LIN {X 0,Y 488.421,Z 680.985,A -85,B 0,C 180,E1 -6398.273,E2 -6398.273} C_VEL
LIN {X 0,Y 488.699,Z 673.076,A -85,B 0,C 180,E1 -6399.52,E2 -6399.52} C_VEL
LIN {X 0,Y 489.009,Z 665.001,A -85,B 0,C 180,E1 -6400.559,E2 -6400.559} C_VEL
LIN {X 0,Y 489.51,Z 655.097,A -85,B 0,C 180,E1 -6401.596,E2 -6401.596} C_VEL
LIN {X 0,Y 489.842,Z 643.67,A -85,B 0,C 180,E1 -6402.557,E2 -6402.557} C_VEL
LIN {X 0,Y 490.248,Z 633.111,A -85,B 0,C 180,E1 -6403.26,E2 -6403.26} C_VEL
LIN {X 0,Y 490.638,Z 620.98,A -85,B 0,C 180,E1 -6403.883,E2 -6403.883} C_VEL
LIN {X 0,Y 490.956,Z 608.45,A -85,B 0,C 180,E1 -6404.349,E2 -6404.349} C_VEL
LIN {X 0,Y 491.208,Z 595.654,A -85,B 0,C 180,E1 -6404.659,E2 -6404.659} C_VEL
LIN {X 0,Y 491.628,Z 499.894,A -85,B 0,C 180,E1 -6406.077,E2 -6406.077} C_VEL
LIN {X 0,Y 489.945,Z 488.116,A -85,B 0,C 180,E1 -6406.322,E2 -6406.322} C_VEL
LIN {X 0,Y 490.166,Z 476.152,A -85,B 0,C 180,E1 -6407.739,E2 -6407.739} C_VEL
LIN {X 0,Y 490.799,Z 452.084,A -85,B 0,C 180,E1 -6410.757,E2 -6410.757} C_VEL
LIN {X 0,Y 491.628,Z 428.446,A -85,B 0,C 180,E1 -6413.807,E2 -6413.807} C_VEL
LIN {X 0,Y 492.314,Z 404.124,A -85,B 0,C 180,E1 -6416.952,E2 -6416.952} C_VEL
LIN {X 0,Y 490.804,Z 396.546,A -85,B 0,C 180,E1 -6418.011,E2 -6418.011} C_VEL
LIN {X 0,Y 488.774,Z 387.78,A -85,B 0,C 180,E1 -6419.267,E2 -6419.267} C_VEL
LIN {X 0,Y 488.706,Z 387.61,A -85,B 0,C 180,E1 -6422.147,E2 -6422.147} C_VEL
LIN {X 0,Y 488.713,Z 387.61,A -85,B 0,C 180,E1 -6425.116,E2 -6425.116} C_VEL
LIN {X 0,Y 488.66,Z 387.615,A -85,B 0,C 180,E1 -6428.202,E2 -6428.202} C_VEL
LIN {X 0,Y 488.696,Z 387.602,A -85,B 0,C 180,E1 -6430.341,E2 -6430.341} C_VEL
LIN {X 0,Y 488.676,Z 387.609,A -85,B 0,C 180,E1 -6433.656,E2 -6433.656} C_VEL
LIN {X 0,Y 488.678,Z 387.61,A -85,B 0,C 180,E1 -6436.344,E2 -6436.344} C_VEL
LIN {X 0,Y 488.707,Z 387.611,A -85,B 0,C 180,E1 -6439.674,E2 -6439.674} C_VEL
LIN {X 0,Y 488.662,Z 387.607,A -85,B 0,C 180,E1 -6442.839,E2 -6442.839} C_VEL
LIN {X 0,Y 488.721,Z 387.604,A -85,B 0,C 180,E1 -6445.886,E2 -6445.886} C_VEL
LIN {X 0,Y 488.693,Z 387.608,A -85,B 0,C 180,E1 -6448.82,E2 -6448.82} C_VEL
LIN {X 0,Y 488.695,Z 387.608,A -85,B 0,C 180,E1 -6451.668,E2 -6451.668} C_VEL
LIN {X 0,Y 488.702,Z 387.606,A -85,B 0,C 180,E1 -6454.959,E2 -6454.959} C_VEL
LIN {X 0,Y 488.7,Z 387.61,A -85,B 0,C 180,E1 -6458.043,E2 -6458.043} C_VEL
LIN {X 0,Y 488.734,Z 387.6,A -85,B 0,C 180,E1 -6460.686,E2 -6460.686} C_VEL
LIN {X 0,Y 488.714,Z 387.607,A -85,B 0,C 180,E1 -6464.143,E2 -6464.143} C_VEL
LIN {X 0,Y 488.725,Z 387.601,A -85,B 0,C 180,E1 -6466.698,E2 -6466.698} C_VEL
LIN {X 0,Y 488.704,Z 387.598,A -85,B 0,C 180,E1 -6469.225,E2 -6469.225} C_VEL
LIN {X 0,Y 488.763,Z 387.606,A -85,B 0,C 180,E1 -6471.733,E2 -6471.733} C_VEL
LIN {X 0,Y 488.816,Z 387.587,A -85,B 0,C 180,E1 -6474.224,E2 -6474.224} C_VEL
LIN {X 0,Y 488.944,Z 387.576,A -85,B 0,C 180,E1 -6477.529,E2 -6477.529} C_VEL
LIN {X 0,Y 488.945,Z 387.578,A -85,B 0,C 180,E1 -6480,E2 -6480} C_VEL
LIN {X 0,Y 488.945,Z 387.566,A -85,B 0,C 180,E1 -6482.471,E2 -6482.471} C_VEL
LIN {X 0,Y 488.814,Z 387.599,A -85,B 0,C 180,E1 -6485.776,E2 -6485.776} C_VEL
LIN {X 0,Y 488.76,Z 387.595,A -85,B 0,C 180,E1 -6488.267,E2 -6488.267} C_VEL
LIN {X 0,Y 488.788,Z 387.596,A -85,B 0,C 180,E1 -6491.613,E2 -6491.613} C_VEL
LIN {X 0,Y 488.723,Z 387.601,A -85,B 0,C 180,E1 -6495.002,E2 -6495.002} C_VEL
LIN {X 0,Y 488.705,Z 387.606,A -85,B 0,C 180,E1 -6498.444,E2 -6498.444} C_VEL
LIN {X 0,Y 488.682,Z 387.608,A -85,B 0,C 180,E1 -6501.072,E2 -6501.072} C_VEL
LIN {X 0,Y 488.667,Z 387.608,A -85,B 0,C 180,E1 -6503.747,E2 -6503.747} C_VEL
LIN {X 0,Y 488.671,Z 387.611,A -85,B 0,C 180,E1 -6506.477,E2 -6506.477} C_VEL
LIN {X 0,Y 488.702,Z 387.6,A -85,B 0,C 180,E1 -6509.272,E2 -6509.272} C_VEL
LIN {X 0,Y 488.692,Z 387.611,A -85,B 0,C 180,E1 -6512.148,E2 -6512.148} C_VEL
LIN {X 0,Y 488.708,Z 387.601,A -85,B 0,C 180,E1 -6515.116,E2 -6515.116} C_VEL
LIN {X 0,Y 488.651,Z 387.612,A -85,B 0,C 180,E1 -6518.203,E2 -6518.203} C_VEL
LIN {X 0,Y 488.644,Z 387.595,A -85,B 0,C 180,E1 -6521.422,E2 -6521.422} C_VEL
LIN {X 0,Y 488.698,Z 387.607,A -85,B 0,C 180,E1 -6524.803,E2 -6524.803} C_VEL
LIN {X 0,Y 488.65,Z 387.613,A -85,B 0,C 180,E1 -6527.469,E2 -6527.469} C_VEL
LIN {X 0,Y 488.671,Z 387.608,A -85,B 0,C 180,E1 -6530.742,E2 -6530.742} C_VEL
LIN {X 0,Y 488.642,Z 387.622,A -85,B 0,C 180,E1 -6533.864,E2 -6533.864} C_VEL
LIN {X 0,Y 488.694,Z 387.611,A -85,B 0,C 180,E1 -6536.523,E2 -6536.523} C_VEL
LIN {X 0,Y 488.666,Z 387.618,A -85,B 0,C 180,E1 -6539.776,E2 -6539.776} C_VEL
LIN {X 0,Y 488.734,Z 387.967,A -85,B 0,C 180,E1 -6540.138,E2 -6540.138} C_VEL
LIN {X 0,Y 492.353,Z 403.874,A -85,B 0,C 180,E1 -6542.467,E2 -6542.467} C_VEL
LIN {X 0,Y 491.871,Z 419.05,A -85,B 0,C 180,E1 -6544.452,E2 -6544.452} C_VEL
LIN {X 0,Y 490.95,Z 442.63,A -85,B 0,C 180,E1 -6547.485,E2 -6547.485} C_VEL
LIN {X 0,Y 490.174,Z 466.628,A -85,B 0,C 180,E1 -6550.527,E2 -6550.527} C_VEL
LIN {X 0,Y 489.479,Z 492.055,A -85,B 0,C 180,E1 -6553.698,E2 -6553.698} C_VEL
LIN {X 0,Y 491.532,Z 510.881,A -85,B 0,C 180,E1 -6554.093,E2 -6554.093} C_VEL
LIN {X 0,Y 490.766,Z 603.473,A -85,B 0,C 180,E1 -6555.566,E2 -6555.566} C_VEL
LIN {X 0,Y 490.386,Z 620.377,A -85,B 0,C 180,E1 -6556.031,E2 -6556.031} C_VEL
LIN {X 0,Y 490.093,Z 633.651,A -85,B 0,C 180,E1 -6556.577,E2 -6556.577} C_VEL
LIN {X 0,Y 489.785,Z 644.595,A -85,B 0,C 180,E1 -6557.191,E2 -6557.191} C_VEL
LIN {X 0,Y 489.453,Z 655.726,A -85,B 0,C 180,E1 -6557.992,E2 -6557.992} C_VEL
LIN {X 0,Y 489.043,Z 666.053,A -85,B 0,C 180,E1 -6558.918,E2 -6558.918} C_VEL
LIN {X 0,Y 488.789,Z 674.567,A -85,B 0,C 180,E1 -6559.855,E2 -6559.855} C_VEL
LIN {X 0,Y 488.508,Z 682.384,A -85,B 0,C 180,E1 -6560.894,E2 -6560.894} C_VEL
LIN {X 0,Y 488.295,Z 689.986,A -85,B 0,C 180,E1 -6562.141,E2 -6562.141} C_VEL
LIN {X 0,Y 488.105,Z 696.43,A -85,B 0,C 180,E1 -6563.465,E2 -6563.465} C_VEL
LIN {X 0,Y 488.086,Z 700.893,A -85,B 0,C 180,E1 -6564.629,E2 -6564.629} C_VEL
LIN {X 0,Y 488.026,Z 704.563,A -85,B 0,C 180,E1 -6565.871,E2 -6565.871} C_VEL
LIN {X 0,Y 488.028,Z 706.453,A -85,B 0,C 180,E1 -6566.698,E2 -6566.698} C_VEL
LIN {X 0,Y 487.974,Z 707.88,A -85,B 0,C 180,E1 -6567.524,E2 -6567.524} C_VEL
LIN {X 0,Y 487.953,Z 708.886,A -85,B 0,C 180,E1 -6568.349,E2 -6568.349} C_VEL
LIN {X 0,Y 487.921,Z 709.721,A -85,B 0,C 180,E1 -6570,E2 -6570} C_VEL
LIN {X 0,Y 487.933,Z 709.501,A -85,B 0,C 180,E1 -6570.825,E2 -6570.825} C_VEL
LIN {X 0,Y 487.958,Z 708.887,A -85,B 0,C 180,E1 -6571.651,E2 -6571.651} C_VEL
LIN {X 0,Y 487.983,Z 707.882,A -85,B 0,C 180,E1 -6572.476,E2 -6572.476} C_VEL
LIN {X 0,Y 488.037,Z 706.455,A -85,B 0,C 180,E1 -6573.302,E2 -6573.302} C_VEL
LIN {X 0,Y 488.016,Z 703.483,A -85,B 0,C 180,E1 -6574.543,E2 -6574.543} C_VEL
LIN {X 0,Y 488.108,Z 699.445,A -85,B 0,C 180,E1 -6575.785,E2 -6575.785} C_VEL
LIN {X 0,Y 488.184,Z 693.211,A -85,B 0,C 180,E1 -6577.237,E2 -6577.237} C_VEL
LIN {X 0,Y 488.42,Z 686.403,A -85,B 0,C 180,E1 -6578.481,E2 -6578.481} C_VEL
LIN {X 0,Y 488.571,Z 679.428,A -85,B 0,C 180,E1 -6579.522,E2 -6579.522} C_VEL
LIN {X 0,Y 488.879,Z 670.989,A -85,B 0,C 180,E1 -6580.561,E2 -6580.561} C_VEL
LIN {X 0,Y 489.254,Z 660.526,A -85,B 0,C 180,E1 -6581.602,E2 -6581.602} C_VEL
LIN {X 0,Y 489.587,Z 650.136,A -85,B 0,C 180,E1 -6582.435,E2 -6582.435} C_VEL
LIN {X 0,Y 489.928,Z 638.639,A -85,B 0,C 180,E1 -6583.163,E2 -6583.163} C_VEL
LIN {X 0,Y 490.285,Z 626.638,A -85,B 0,C 180,E1 -6583.734,E2 -6583.734} C_VEL
LIN {X 0,Y 490.503,Z 614.471,A -85,B 0,C 180,E1 -6584.151,E2 -6584.151} C_VEL
LIN {X 0,Y 490.732,Z 602.483,A -85,B 0,C 180,E1 -6584.409,E2 -6584.409} C_VEL
LIN {X 0,Y 491.382,Z 509.881,A -85,B 0,C 180,E1 -6585.871,E2 -6585.871} C_VEL
LIN {X 0,Y 489.25,Z 488.746,A -85,B 0,C 180,E1 -6586.327,E2 -6586.327} C_VEL
LIN {X 0,Y 489.772,Z 466.119,A -85,B 0,C 180,E1 -6589.098,E2 -6589.098} C_VEL
LIN {X 0,Y 490.419,Z 442.199,A -85,B 0,C 180,E1 -6592.097,E2 -6592.097} C_VEL
LIN {X 0,Y 491.22,Z 418.158,A -85,B 0,C 180,E1 -6595.191,E2 -6595.191} C_VEL
LIN {X 0,Y 491.802,Z 402.9,A -85,B 0,C 180,E1 -6597.212,E2 -6597.212} C_VEL
LIN {X 0,Y 489.495,Z 391.112,A -85,B 0,C 180,E1 -6598.972,E2 -6598.972} C_VEL
LIN {X 0,Y 488.701,Z 387.728,A -85,B 0,C 180,E1 -6599.538,E2 -6599.538} C_VEL
LIN {X 0,Y 488.679,Z 387.616,A -85,B 0,C 180,E1 -6602.149,E2 -6602.149} C_VEL
LIN {X 0,Y 488.696,Z 387.611,A -85,B 0,C 180,E1 -6605.117,E2 -6605.117} C_VEL
LIN {X 0,Y 488.65,Z 387.619,A -85,B 0,C 180,E1 -6608.203,E2 -6608.203} C_VEL
LIN {X 0,Y 488.644,Z 387.618,A -85,B 0,C 180,E1 -6611.422,E2 -6611.422} C_VEL
LIN {X 0,Y 488.702,Z 387.608,A -85,B 0,C 180,E1 -6614.803,E2 -6614.803} C_VEL
LIN {X 0,Y 488.651,Z 387.617,A -85,B 0,C 180,E1 -6617.47,E2 -6617.47} C_VEL
LIN {X 0,Y 488.705,Z 387.612,A -85,B 0,C 180,E1 -6619.674,E2 -6619.674} C_VEL
LIN {X 0,Y 488.662,Z 387.613,A -85,B 0,C 180,E1 -6622.839,E2 -6622.839} C_VEL
LIN {X 0,Y 488.725,Z 387.609,A -85,B 0,C 180,E1 -6625.887,E2 -6625.887} C_VEL
LIN {X 0,Y 488.694,Z 387.61,A -85,B 0,C 180,E1 -6628.82,E2 -6628.82} C_VEL
LIN {X 0,Y 488.714,Z 387.612,A -85,B 0,C 180,E1 -6631.669,E2 -6631.669} C_VEL
LIN {X 0,Y 488.707,Z 387.606,A -85,B 0,C 180,E1 -6634.442,E2 -6634.442} C_VEL
LIN {X 0,Y 488.724,Z 387.61,A -85,B 0,C 180,E1 -6637.153,E2 -6637.153} C_VEL
LIN {X 0,Y 488.728,Z 387.609,A -85,B 0,C 180,E1 -6639.811,E2 -6639.811} C_VEL
LIN {X 0,Y 488.718,Z 387.61,A -85,B 0,C 180,E1 -6642.423,E2 -6642.423} C_VEL
LIN {X 0,Y 488.774,Z 387.749,A -85,B 0,C 180,E1 -6644.092,E2 -6644.092} C_VEL
LIN {X 0,Y 488.957,Z 388.568,A -85,B 0,C 180,E1 -6644.226,E2 -6644.226} C_VEL
LIN {X 0,Y 491.703,Z 396.705,A -85,B 0,C 180,E1 -6644.497,E2 -6644.497} C_VEL
LIN {X 0,Y 491.048,Z 471.478,A -85,B 0,C 180,E1 -6645.76,E2 -6645.76} C_VEL
LIN {X 0,Y 490.918,Z 485.433,A -85,B 0,C 180,E1 -6646.178,E2 -6646.178} C_VEL
LIN {X 0,Y 490.785,Z 498.232,A -85,B 0,C 180,E1 -6646.755,E2 -6646.755} C_VEL
LIN {X 0,Y 490.578,Z 510.162,A -85,B 0,C 180,E1 -6647.475,E2 -6647.475} C_VEL
LIN {X 0,Y 490.245,Z 521.111,A -85,B 0,C 180,E1 -6648.317,E2 -6648.317} C_VEL
LIN {X 0,Y 489.959,Z 530.794,A -85,B 0,C 180,E1 -6649.253,E2 -6649.253} C_VEL
LIN {X 0,Y 489.7,Z 539.557,A -85,B 0,C 180,E1 -6650.292,E2 -6650.292} C_VEL
LIN {X 0,Y 489.412,Z 546.759,A -85,B 0,C 180,E1 -6651.328,E2 -6651.328} C_VEL
LIN {X 0,Y 489.082,Z 553.808,A -85,B 0,C 180,E1 -6652.569,E2 -6652.569} C_VEL
LIN {X 0,Y 488.992,Z 559.358,A -85,B 0,C 180,E1 -6653.812,E2 -6653.812} C_VEL
LIN {X 0,Y 488.733,Z 563.713,A -85,B 0,C 180,E1 -6655.05,E2 -6655.05} C_VEL
LIN {X 0,Y 488.65,Z 565.979,A -85,B 0,C 180,E1 -6655.876,E2 -6655.876} C_VEL
LIN {X 0,Y 488.703,Z 567.797,A -85,B 0,C 180,E1 -6656.702,E2 -6656.702} C_VEL
LIN {X 0,Y 488.561,Z 569.208,A -85,B 0,C 180,E1 -6657.527,E2 -6657.527} C_VEL
LIN {X 0,Y 488.58,Z 570.15,A -85,B 0,C 180,E1 -6658.351,E2 -6658.351} C_VEL
LIN {X 0,Y 488.487,Z 570.885,A -85,B 0,C 180,E1 -6660,E2 -6660} C_VEL
LIN {X 0,Y 488.504,Z 570.624,A -85,B 0,C 180,E1 -6660.824,E2 -6660.824} C_VEL
LIN {X 0,Y 488.438,Z 569.968,A -85,B 0,C 180,E1 -6661.649,E2 -6661.649} C_VEL
LIN {X 0,Y 488.535,Z 568.897,A -85,B 0,C 180,E1 -6662.474,E2 -6662.474} C_VEL
LIN {X 0,Y 488.495,Z 567.446,A -85,B 0,C 180,E1 -6663.299,E2 -6663.299} C_VEL
LIN {X 0,Y 488.648,Z 564.404,A -85,B 0,C 180,E1 -6664.537,E2 -6664.537} C_VEL
LIN {X 0,Y 488.745,Z 560.322,A -85,B 0,C 180,E1 -6665.777,E2 -6665.777} C_VEL
LIN {X 0,Y 488.981,Z 554.834,A -85,B 0,C 180,E1 -6667.061,E2 -6667.061} C_VEL
LIN {X 0,Y 489.212,Z 547.178,A -85,B 0,C 180,E1 -6668.468,E2 -6668.468} C_VEL
LIN {X 0,Y 489.485,Z 540.175,A -85,B 0,C 180,E1 -6669.504,E2 -6669.504} C_VEL
LIN {X 0,Y 489.681,Z 531.737,A -85,B 0,C 180,E1 -6670.544,E2 -6670.544} C_VEL
LIN {X 0,Y 489.989,Z 521.287,A -85,B 0,C 180,E1 -6671.584,E2 -6671.584} C_VEL
LIN {X 0,Y 490.392,Z 509.565,A -85,B 0,C 180,E1 -6672.512,E2 -6672.512} C_VEL
LIN {X 0,Y 490.542,Z 497.636,A -85,B 0,C 180,E1 -6673.252,E2 -6673.252} C_VEL
LIN {X 0,Y 490.776,Z 485.334,A -85,B 0,C 180,E1 -6673.826,E2 -6673.826} C_VEL
LIN {X 0,Y 490.962,Z 472.814,A -85,B 0,C 180,E1 -6674.243,E2 -6674.243} C_VEL
LIN {X 0,Y 491.012,Z 458.482,A -85,B 0,C 180,E1 -6674.533,E2 -6674.533} C_VEL
LIN {X 0,Y 491.417,Z 395.815,A -85,B 0,C 180,E1 -6675.535,E2 -6675.535} C_VEL
LIN {X 0,Y 488.913,Z 388.41,A -85,B 0,C 180,E1 -6675.764,E2 -6675.764} C_VEL
LIN {X 0,Y 488.774,Z 387.692,A -85,B 0,C 180,E1 -6675.908,E2 -6675.908} C_VEL
LIN {X 0,Y 488.745,Z 387.605,A -85,B 0,C 180,E1 -6679.313,E2 -6679.313} C_VEL
LIN {X 0,Y 488.701,Z 387.608,A -85,B 0,C 180,E1 -6681.957,E2 -6681.957} C_VEL
LIN {X 0,Y 488.734,Z 387.607,A -85,B 0,C 180,E1 -6685.049,E2 -6685.049} C_VEL
LIN {X 0,Y 488.709,Z 387.603,A -85,B 0,C 180,E1 -6687.399,E2 -6687.399} C_VEL
LIN {X 0,Y 488.712,Z 387.605,A -85,B 0,C 180,E1 -6690.363,E2 -6690.363} C_VEL
LIN {X 0,Y 488.732,Z 387.597,A -85,B 0,C 180,E1 -6693.483,E2 -6693.483} C_VEL
LIN {X 0,Y 488.683,Z 387.612,A -85,B 0,C 180,E1 -6696.354,E2 -6696.354} C_VEL
LIN {X 0,Y 488.703,Z 387.608,A -85,B 0,C 180,E1 -6699.254,E2 -6699.254} C_VEL
LIN {X 0,Y 488.69,Z 387.61,A -85,B 0,C 180,E1 -6702.526,E2 -6702.526} C_VEL
LIN {X 0,Y 488.703,Z 387.606,A -85,B 0,C 180,E1 -6705.197,E2 -6705.197} C_VEL
LIN {X 0,Y 488.697,Z 387.612,A -85,B 0,C 180,E1 -6708.583,E2 -6708.583} C_VEL
LIN {X 0,Y 488.703,Z 387.6,A -85,B 0,C 180,E1 -6710.948,E2 -6710.948} C_VEL
LIN {X 0,Y 488.666,Z 387.613,A -85,B 0,C 180,E1 -6713.462,E2 -6713.462} C_VEL
LIN {X 0,Y 488.026,Z 387.695,A -85,B 0,C 180,E1 -6714.15,E2 -6714.15} C_VEL
LIN {X 0,Y 485.191,Z 388.045,A -85,B 0,C 180,E1 -6715.267,E2 -6715.267} C_VEL
LIN {X 0,Y 482.782,Z 388.347,A -85,B 0,C 180,E1 -6716.167,E2 -6716.167} C_VEL
LIN {X 0,Y 481.751,Z 388.474,A -85,B 0,C 180,E1 -6716.863,E2 -6716.863} C_VEL
LIN {X 0,Y 481.67,Z 388.481,A -85,B 0,C 180,E1 -6717.098,E2 -6717.098} C_VEL
LIN {X 0,Y 481.734,Z 388.669,A -85,B 0,C 180,E1 -6720.575,E2 -6720.575} C_VEL
LIN {X 0,Y 485.358,Z 404.631,A -85,B 0,C 180,E1 -6722.863,E2 -6722.863} C_VEL
LIN {X 0,Y 485.19,Z 415.109,A -85,B 0,C 180,E1 -6724.243,E2 -6724.243} C_VEL
LIN {X 0,Y 484.486,Z 435.748,A -85,B 0,C 180,E1 -6726.942,E2 -6726.942} C_VEL
LIN {X 0,Y 483.714,Z 457.932,A -85,B 0,C 180,E1 -6729.814,E2 -6729.814} C_VEL
LIN {X 0,Y 483.09,Z 482.393,A -85,B 0,C 180,E1 -6732.867,E2 -6732.867} C_VEL
LIN {X 0,Y 482.979,Z 488.109,A -85,B 0,C 180,E1 -6733.531,E2 -6733.531} C_VEL
LIN {X 0,Y 484.947,Z 502.633,A -85,B 0,C 180,E1 -6733.829,E2 -6733.829} C_VEL
LIN {X 0,Y 484.243,Z 598.949,A -85,B 0,C 180,E1 -6735.287,E2 -6735.287} C_VEL
LIN {X 0,Y 483.985,Z 612.191,A -85,B 0,C 180,E1 -6735.655,E2 -6735.655} C_VEL
LIN {X 0,Y 483.6,Z 624.672,A -85,B 0,C 180,E1 -6736.18,E2 -6736.18} C_VEL
LIN {X 0,Y 483.21,Z 636.877,A -85,B 0,C 180,E1 -6736.873,E2 -6736.873} C_VEL
LIN {X 0,Y 482.826,Z 648.198,A -85,B 0,C 180,E1 -6737.709,E2 -6737.709} C_VEL
LIN {X 0,Y 482.267,Z 659.494,A -85,B 0,C 180,E1 -6738.76,E2 -6738.76} C_VEL
LIN {X 0,Y 481.957,Z 667.756,A -85,B 0,C 180,E1 -6739.71,E2 -6739.71} C_VEL
LIN {X 0,Y 481.604,Z 675.394,A -85,B 0,C 180,E1 -6740.763,E2 -6740.763} C_VEL
LIN {X 0,Y 481.31,Z 682.842,A -85,B 0,C 180,E1 -6742.026,E2 -6742.026} C_VEL
LIN {X 0,Y 481.117,Z 689.192,A -85,B 0,C 180,E1 -6743.377,E2 -6743.377} C_VEL
LIN {X 0,Y 481.009,Z 693.557,A -85,B 0,C 180,E1 -6744.55,E2 -6744.55} C_VEL
LIN {X 0,Y 480.88,Z 697.183,A -85,B 0,C 180,E1 -6745.81,E2 -6745.81} C_VEL
LIN {X 0,Y 480.899,Z 699.049,A -85,B 0,C 180,E1 -6746.649,E2 -6746.649} C_VEL
LIN {X 0,Y 480.824,Z 700.479,A -85,B 0,C 180,E1 -6747.487,E2 -6747.487} C_VEL
LIN {X 0,Y 480.76,Z 702.099,A -85,B 0,C 180,E1 -6749.163,E2 -6749.163} C_VEL
LIN {X 0,Y 480.743,Z 702.337,A -85,B 0,C 180,E1 -6750,E2 -6750} C_VEL
LIN {X 0,Y 480.76,Z 702.149,A -85,B 0,C 180,E1 -6750.838,E2 -6750.838} C_VEL
LIN {X 0,Y 480.824,Z 700.596,A -85,B 0,C 180,E1 -6752.513,E2 -6752.513} C_VEL
LIN {X 0,Y 480.899,Z 699.231,A -85,B 0,C 180,E1 -6753.351,E2 -6753.351} C_VEL
LIN {X 0,Y 480.868,Z 696.358,A -85,B 0,C 180,E1 -6754.611,E2 -6754.611} C_VEL
LIN {X 0,Y 481.022,Z 692.455,A -85,B 0,C 180,E1 -6755.87,E2 -6755.87} C_VEL
LIN {X 0,Y 481.099,Z 687.4,A -85,B 0,C 180,E1 -6757.133,E2 -6757.133} C_VEL
LIN {X 0,Y 481.383,Z 681.027,A -85,B 0,C 180,E1 -6758.395,E2 -6758.395} C_VEL
LIN {X 0,Y 481.684,Z 673.114,A -85,B 0,C 180,E1 -6759.66,E2 -6759.66} C_VEL
LIN {X 0,Y 482.019,Z 665.035,A -85,B 0,C 180,E1 -6760.714,E2 -6760.714} C_VEL
LIN {X 0,Y 482.552,Z 655.123,A -85,B 0,C 180,E1 -6761.765,E2 -6761.765} C_VEL
LIN {X 0,Y 482.883,Z 643.885,A -85,B 0,C 180,E1 -6762.725,E2 -6762.725} C_VEL
LIN {X 0,Y 483.322,Z 633.118,A -85,B 0,C 180,E1 -6763.454,E2 -6763.454} C_VEL
LIN {X 0,Y 483.757,Z 620.964,A -85,B 0,C 180,E1 -6764.084,E2 -6764.084} C_VEL
LIN {X 0,Y 484.084,Z 608.403,A -85,B 0,C 180,E1 -6764.557,E2 -6764.557} C_VEL
LIN {X 0,Y 484.342,Z 595.515,A -85,B 0,C 180,E1 -6764.872,E2 -6764.872} C_VEL
LIN {X 0,Y 484.844,Z 500.841,A -85,B 0,C 180,E1 -6766.292,E2 -6766.292} C_VEL
LIN {X 0,Y 483,Z 487.823,A -85,B 0,C 180,E1 -6766.574,E2 -6766.574} C_VEL
LIN {X 0,Y 483.443,Z 467.2,A -85,B 0,C 180,E1 -6769.102,E2 -6769.102} C_VEL
LIN {X 0,Y 484.299,Z 441.592,A -85,B 0,C 180,E1 -6772.392,E2 -6772.392} C_VEL
LIN {X 0,Y 485.016,Z 421.047,A -85,B 0,C 180,E1 -6775.078,E2 -6775.078} C_VEL
LIN {X 0,Y 485.444,Z 405.294,A -85,B 0,C 180,E1 -6777.132,E2 -6777.132} C_VEL
LIN {X 0,Y 482.041,Z 389.921,A -85,B 0,C 180,E1 -6779.316,E2 -6779.316} C_VEL
LIN {X 0,Y 481.698,Z 388.508,A -85,B 0,C 180,E1 -6779.589,E2 -6779.589} C_VEL
LIN {X 0,Y 481.674,Z 388.486,A -85,B 0,C 180,E1 -6782.674,E2 -6782.674} C_VEL
LIN {X 0,Y 481.624,Z 388.492,A -85,B 0,C 180,E1 -6785.711,E2 -6785.711} C_VEL
LIN {X 0,Y 481.635,Z 388.489,A -85,B 0,C 180,E1 -6788.863,E2 -6788.863} C_VEL
LIN {X 0,Y 481.624,Z 388.494,A -85,B 0,C 180,E1 -6791.909,E2 -6791.909} C_VEL
LIN {X 0,Y 481.657,Z 388.474,A -85,B 0,C 180,E1 -6794.458,E2 -6794.458} C_VEL
LIN {X 0,Y 481.628,Z 388.494,A -85,B 0,C 180,E1 -6797.837,E2 -6797.837} C_VEL
LIN {X 0,Y 481.659,Z 388.487,A -85,B 0,C 180,E1 -6801.14,E2 -6801.14} C_VEL
LIN {X 0,Y 481.658,Z 388.484,A -85,B 0,C 180,E1 -6804.797,E2 -6804.797} C_VEL
LIN {X 0,Y 481.653,Z 388.49,A -85,B 0,C 180,E1 -6807.812,E2 -6807.812} C_VEL
LIN {X 0,Y 481.669,Z 388.48,A -85,B 0,C 180,E1 -6810.258,E2 -6810.258} C_VEL
LIN {X 0,Y 481.662,Z 388.484,A -85,B 0,C 180,E1 -6813.107,E2 -6813.107} C_VEL
LIN {X 0,Y 481.652,Z 388.483,A -85,B 0,C 180,E1 -6815.885,E2 -6815.885} C_VEL
LIN {X 0,Y 481.707,Z 388.478,A -85,B 0,C 180,E1 -6819.028,E2 -6819.028} C_VEL
LIN {X 0,Y 481.675,Z 388.477,A -85,B 0,C 180,E1 -6822.157,E2 -6822.157} C_VEL
LIN {X 0,Y 481.734,Z 388.474,A -85,B 0,C 180,E1 -6824.775,E2 -6824.775} C_VEL
LIN {X 0,Y 481.739,Z 388.465,A -85,B 0,C 180,E1 -6828.215,E2 -6828.215} C_VEL
LIN {X 0,Y 481.722,Z 388.481,A -85,B 0,C 180,E1 -6831.611,E2 -6831.611} C_VEL
LIN {X 0,Y 481.778,Z 388.464,A -85,B 0,C 180,E1 -6834.139,E2 -6834.139} C_VEL
LIN {X 0,Y 481.91,Z 388.452,A -85,B 0,C 180,E1 -6837.492,E2 -6837.492} C_VEL
LIN {X 0,Y 481.914,Z 388.453,A -85,B 0,C 180,E1 -6840,E2 -6840} C_VEL
LIN {X 0,Y 481.91,Z 388.442,A -85,B 0,C 180,E1 -6842.508,E2 -6842.508} C_VEL
LIN {X 0,Y 481.776,Z 388.476,A -85,B 0,C 180,E1 -6845.861,E2 -6845.861} C_VEL
LIN {X 0,Y 481.719,Z 388.47,A -85,B 0,C 180,E1 -6848.389,E2 -6848.389} C_VEL
LIN {X 0,Y 481.739,Z 388.476,A -85,B 0,C 180,E1 -6851.785,E2 -6851.785} C_VEL
LIN {X 0,Y 481.696,Z 388.477,A -85,B 0,C 180,E1 -6855.226,E2 -6855.226} C_VEL
LIN {X 0,Y 481.639,Z 388.485,A -85,B 0,C 180,E1 -6858.725,E2 -6858.725} C_VEL
LIN {X 0,Y 481.628,Z 388.489,A -85,B 0,C 180,E1 -6861.396,E2 -6861.396} C_VEL
LIN {X 0,Y 481.646,Z 388.488,A -85,B 0,C 180,E1 -6864.115,E2 -6864.115} C_VEL
LIN {X 0,Y 481.645,Z 388.485,A -85,B 0,C 180,E1 -6867.114,E2 -6867.114} C_VEL
LIN {X 0,Y 481.667,Z 388.481,A -85,B 0,C 180,E1 -6869.742,E2 -6869.742} C_VEL
LIN {X 0,Y 481.65,Z 388.484,A -85,B 0,C 180,E1 -6872.676,E2 -6872.676} C_VEL
LIN {X 0,Y 481.651,Z 388.48,A -85,B 0,C 180,E1 -6875.202,E2 -6875.202} C_VEL
LIN {X 0,Y 481.628,Z 388.49,A -85,B 0,C 180,E1 -6878.002,E2 -6878.002} C_VEL
LIN {X 0,Y 481.605,Z 388.471,A -85,B 0,C 180,E1 -6881.047,E2 -6881.047} C_VEL
LIN {X 0,Y 481.652,Z 388.486,A -85,B 0,C 180,E1 -6884.458,E2 -6884.458} C_VEL
LIN {X 0,Y 481.614,Z 388.486,A -85,B 0,C 180,E1 -6886.856,E2 -6886.856} C_VEL
LIN {X 0,Y 481.63,Z 388.481,A -85,B 0,C 180,E1 -6890.054,E2 -6890.054} C_VEL
LIN {X 0,Y 481.605,Z 388.492,A -85,B 0,C 180,E1 -6893.251,E2 -6893.251} C_VEL
LIN {X 0,Y 481.672,Z 388.488,A -85,B 0,C 180,E1 -6896.327,E2 -6896.327} C_VEL
LIN {X 0,Y 481.653,Z 388.627,A -85,B 0,C 180,E1 -6899.85,E2 -6899.85} C_VEL
LIN {X 0,Y 485.352,Z 404.76,A -85,B 0,C 180,E1 -6902.264,E2 -6902.264} C_VEL
LIN {X 0,Y 485.383,Z 410.93,A -85,B 0,C 180,E1 -6903.097,E2 -6903.097} C_VEL
LIN {X 0,Y 484.38,Z 433.648,A -85,B 0,C 180,E1 -6906.076,E2 -6906.076} C_VEL
LIN {X 0,Y 483.557,Z 455.568,A -85,B 0,C 180,E1 -6908.917,E2 -6908.917} C_VEL
LIN {X 0,Y 482.786,Z 479.5,A -85,B 0,C 180,E1 -6911.98,E2 -6911.98} C_VEL
LIN {X 0,Y 482.489,Z 491.243,A -85,B 0,C 180,E1 -6913.455,E2 -6913.455} C_VEL
LIN {X 0,Y 484.687,Z 511.595,A -85,B 0,C 180,E1 -6913.889,E2 -6913.889} C_VEL
LIN {X 0,Y 483.848,Z 603.001,A -85,B 0,C 180,E1 -6915.382,E2 -6915.382} C_VEL
LIN {X 0,Y 483.576,Z 617.223,A -85,B 0,C 180,E1 -6915.723,E2 -6915.723} C_VEL
LIN {X 0,Y 483.298,Z 629.158,A -85,B 0,C 180,E1 -6916.17,E2 -6916.17} C_VEL
LIN {X 0,Y 482.999,Z 640.776,A -85,B 0,C 180,E1 -6916.773,E2 -6916.773} C_VEL
LIN {X 0,Y 482.61,Z 652.01,A -85,B 0,C 180,E1 -6917.526,E2 -6917.526} C_VEL
LIN {X 0,Y 482.15,Z 662.815,A -85,B 0,C 180,E1 -6918.438,E2 -6918.438} C_VEL
LIN {X 0,Y 481.808,Z 672.749,A -85,B 0,C 180,E1 -6919.494,E2 -6919.494} C_VEL
LIN {X 0,Y 481.495,Z 680.865,A -85,B 0,C 180,E1 -6920.549,E2 -6920.549} C_VEL
LIN {X 0,Y 481.265,Z 688.806,A -85,B 0,C 180,E1 -6921.814,E2 -6921.814} C_VEL
LIN {X 0,Y 481.096,Z 694.165,A -85,B 0,C 180,E1 -6922.867,E2 -6922.867} C_VEL
LIN {X 0,Y 481.014,Z 699.394,A -85,B 0,C 180,E1 -6924.13,E2 -6924.13} C_VEL
LIN {X 0,Y 480.904,Z 703.429,A -85,B 0,C 180,E1 -6925.39,E2 -6925.39} C_VEL
LIN {X 0,Y 480.951,Z 706.4,A -85,B 0,C 180,E1 -6926.649,E2 -6926.649} C_VEL
LIN {X 0,Y 480.885,Z 707.827,A -85,B 0,C 180,E1 -6927.487,E2 -6927.487} C_VEL
LIN {X 0,Y 480.88,Z 708.832,A -85,B 0,C 180,E1 -6928.325,E2 -6928.325} C_VEL
LIN {X 0,Y 480.839,Z 709.667,A -85,B 0,C 180,E1 -6930,E2 -6930} C_VEL
LIN {X 0,Y 480.853,Z 709.447,A -85,B 0,C 180,E1 -6930.837,E2 -6930.837} C_VEL
LIN {X 0,Y 480.885,Z 708.833,A -85,B 0,C 180,E1 -6931.675,E2 -6931.675} C_VEL
LIN {X 0,Y 480.894,Z 707.828,A -85,B 0,C 180,E1 -6932.513,E2 -6932.513} C_VEL
LIN {X 0,Y 480.96,Z 706.402,A -85,B 0,C 180,E1 -6933.351,E2 -6933.351} C_VEL
LIN {X 0,Y 480.929,Z 703.431,A -85,B 0,C 180,E1 -6934.61,E2 -6934.61} C_VEL
LIN {X 0,Y 481.025,Z 699.395,A -85,B 0,C 180,E1 -6935.87,E2 -6935.87} C_VEL
LIN {X 0,Y 481.114,Z 693.163,A -85,B 0,C 180,E1 -6937.343,E2 -6937.343} C_VEL
LIN {X 0,Y 481.37,Z 686.358,A -85,B 0,C 180,E1 -6938.607,E2 -6938.607} C_VEL
LIN {X 0,Y 481.549,Z 679.385,A -85,B 0,C 180,E1 -6939.662,E2 -6939.662} C_VEL
LIN {X 0,Y 481.881,Z 670.951,A -85,B 0,C 180,E1 -6940.717,E2 -6940.717} C_VEL
LIN {X 0,Y 482.299,Z 660.493,A -85,B 0,C 180,E1 -6941.771,E2 -6941.771} C_VEL
LIN {X 0,Y 482.668,Z 649.12,A -85,B 0,C 180,E1 -6942.69,E2 -6942.69} C_VEL
LIN {X 0,Y 483.016,Z 638.626,A -85,B 0,C 180,E1 -6943.355,E2 -6943.355} C_VEL
LIN {X 0,Y 483.376,Z 626.642,A -85,B 0,C 180,E1 -6943.934,E2 -6943.934} C_VEL
LIN {X 0,Y 483.699,Z 613.6,A -85,B 0,C 180,E1 -6944.381,E2 -6944.381} C_VEL
LIN {X 0,Y 483.845,Z 600.94,A -85,B 0,C 180,E1 -6944.645,E2 -6944.645} C_VEL
LIN {X 0,Y 484.236,Z 540.25,A -85,B 0,C 180,E1 -6945.58,E2 -6945.58} C_VEL
LIN {X 0,Y 484.47,Z 510.049,A -85,B 0,C 180,E1 -6946.089,E2 -6946.089} C_VEL
LIN {X 0,Y 482.265,Z 487.739,A -85,B 0,C 180,E1 -6946.564,E2 -6946.564} C_VEL
LIN {X 0,Y 482.785,Z 465.338,A -85,B 0,C 180,E1 -6949.349,E2 -6949.349} C_VEL
LIN {X 0,Y 483.433,Z 443.001,A -85,B 0,C 180,E1 -6952.209,E2 -6952.209} C_VEL
LIN {X 0,Y 484.313,Z 419.119,A -85,B 0,C 180,E1 -6955.346,E2 -6955.346} C_VEL
LIN {X 0,Y 484.918,Z 404.002,A -85,B 0,C 180,E1 -6957.397,E2 -6957.397} C_VEL
LIN {X 0,Y 482.329,Z 391.5,A -85,B 0,C 180,E1 -6959.328,E2 -6959.328} C_VEL
LIN {X 0,Y 481.644,Z 388.609,A -85,B 0,C 180,E1 -6959.834,E2 -6959.834} C_VEL
LIN {X 0,Y 481.634,Z 388.491,A -85,B 0,C 180,E1 -6962.677,E2 -6962.677} C_VEL
LIN {X 0,Y 481.64,Z 388.491,A -85,B 0,C 180,E1 -6965.2,E2 -6965.2} C_VEL
LIN {X 0,Y 481.626,Z 388.494,A -85,B 0,C 180,E1 -6968.003,E2 -6968.003} C_VEL
LIN {X 0,Y 481.605,Z 388.492,A -85,B 0,C 180,E1 -6971.047,E2 -6971.047} C_VEL
LIN {X 0,Y 481.655,Z 388.487,A -85,B 0,C 180,E1 -6974.458,E2 -6974.458} C_VEL
LIN {X 0,Y 481.616,Z 388.489,A -85,B 0,C 180,E1 -6976.855,E2 -6976.855} C_VEL
LIN {X 0,Y 481.657,Z 388.488,A -85,B 0,C 180,E1 -6980.057,E2 -6980.057} C_VEL
LIN {X 0,Y 481.619,Z 388.495,A -85,B 0,C 180,E1 -6983.378,E2 -6983.378} C_VEL
LIN {X 0,Y 481.678,Z 388.483,A -85,B 0,C 180,E1 -6986.327,E2 -6986.327} C_VEL
LIN {X 0,Y 481.653,Z 388.49,A -85,B 0,C 180,E1 -6989.417,E2 -6989.417} C_VEL
LIN {X 0,Y 481.669,Z 388.485,A -85,B 0,C 180,E1 -6992.166,E2 -6992.166} C_VEL
LIN {X 0,Y 481.68,Z 388.484,A -85,B 0,C 180,E1 -6994.968,E2 -6994.968} C_VEL
LIN {X 0,Y 481.652,Z 388.49,A -85,B 0,C 180,E1 -6997.705,E2 -6997.705} C_VEL
LIN {X 0,Y 481.708,Z 388.482,A -85,B 0,C 180,E1 -7000.393,E2 -7000.393} C_VEL
LIN {X 0,Y 481.73,Z 388.57,A -85,B 0,C 180,E1 -7003.798,E2 -7003.798} C_VEL
LIN {X 0,Y 481.937,Z 389.565,A -85,B 0,C 180,E1 -7003.969,E2 -7003.969} C_VEL
LIN {X 0,Y 484.844,Z 397.313,A -85,B 0,C 180,E1 -7004.241,E2 -7004.241} C_VEL
LIN {X 0,Y 484.209,Z 472.379,A -85,B 0,C 180,E1 -7005.554,E2 -7005.554} C_VEL
LIN {X 0,Y 484.096,Z 486.325,A -85,B 0,C 180,E1 -7005.98,E2 -7005.98} C_VEL
LIN {X 0,Y 483.977,Z 498.198,A -85,B 0,C 180,E1 -7006.512,E2 -7006.512} C_VEL
LIN {X 0,Y 483.757,Z 509.559,A -85,B 0,C 180,E1 -7007.186,E2 -7007.186} C_VEL
LIN {X 0,Y 483.467,Z 520.893,A -85,B 0,C 180,E1 -7008.045,E2 -7008.045} C_VEL
LIN {X 0,Y 483.104,Z 529.88,A -85,B 0,C 180,E1 -7008.886,E2 -7008.886} C_VEL
LIN {X 0,Y 482.839,Z 539.033,A -85,B 0,C 180,E1 -7009.941,E2 -7009.941} C_VEL
LIN {X 0,Y 482.503,Z 546.521,A -85,B 0,C 180,E1 -7010.991,E2 -7010.991} C_VEL
LIN {X 0,Y 482.178,Z 554.405,A -85,B 0,C 180,E1 -7012.368,E2 -7012.368} C_VEL
LIN {X 0,Y 482.018,Z 560.443,A -85,B 0,C 180,E1 -7013.722,E2 -7013.722} C_VEL
LIN {X 0,Y 481.741,Z 564.785,A -85,B 0,C 180,E1 -7014.978,E2 -7014.978} C_VEL
LIN {X 0,Y 481.649,Z 567.042,A -85,B 0,C 180,E1 -7015.816,E2 -7015.816} C_VEL
LIN {X 0,Y 481.699,Z 568.849,A -85,B 0,C 180,E1 -7016.654,E2 -7016.654} C_VEL
LIN {X 0,Y 481.55,Z 570.252,A -85,B 0,C 180,E1 -7017.491,E2 -7017.491} C_VEL
LIN {X 0,Y 481.567,Z 571.181,A -85,B 0,C 180,E1 -7018.327,E2 -7018.327} C_VEL
LIN {X 0,Y 481.468,Z 571.896,A -85,B 0,C 180,E1 -7020,E2 -7020} C_VEL
LIN {X 0,Y 481.485,Z 571.621,A -85,B 0,C 180,E1 -7020.836,E2 -7020.836} C_VEL
LIN {X 0,Y 481.415,Z 570.948,A -85,B 0,C 180,E1 -7021.673,E2 -7021.673} C_VEL
LIN {X 0,Y 481.519,Z 569.863,A -85,B 0,C 180,E1 -7022.51,E2 -7022.51} C_VEL
LIN {X 0,Y 481.47,Z 568.396,A -85,B 0,C 180,E1 -7023.347,E2 -7023.347} C_VEL
LIN {X 0,Y 481.634,Z 565.322,A -85,B 0,C 180,E1 -7024.603,E2 -7024.603} C_VEL
LIN {X 0,Y 481.749,Z 561.2,A -85,B 0,C 180,E1 -7025.861,E2 -7025.861} C_VEL
LIN {X 0,Y 482.007,Z 555.667,A -85,B 0,C 180,E1 -7027.163,E2 -7027.163} C_VEL
LIN {X 0,Y 482.236,Z 547.955,A -85,B 0,C 180,E1 -7028.591,E2 -7028.591} C_VEL
LIN {X 0,Y 482.533,Z 540.898,A -85,B 0,C 180,E1 -7029.642,E2 -7029.642} C_VEL
LIN {X 0,Y 482.741,Z 532.396,A -85,B 0,C 180,E1 -7030.697,E2 -7030.697} C_VEL
LIN {X 0,Y 483.066,Z 521.847,A -85,B 0,C 180,E1 -7031.752,E2 -7031.752} C_VEL
LIN {X 0,Y 483.476,Z 510.259,A -85,B 0,C 180,E1 -7032.678,E2 -7032.678} C_VEL
LIN {X 0,Y 483.652,Z 499.264,A -85,B 0,C 180,E1 -7033.373,E2 -7033.373} C_VEL
LIN {X 0,Y 483.882,Z 486.744,A -85,B 0,C 180,E1 -7033.973,E2 -7033.973} C_VEL
LIN {X 0,Y 484.061,Z 473.539,A -85,B 0,C 180,E1 -7034.424,E2 -7034.424} C_VEL
LIN {X 0,Y 484.124,Z 459.172,A -85,B 0,C 180,E1 -7034.717,E2 -7034.717} C_VEL
LIN {X 0,Y 484.495,Z 396.973,A -85,B 0,C 180,E1 -7035.732,E2 -7035.732} C_VEL
LIN {X 0,Y 481.903,Z 389.412,A -85,B 0,C 180,E1 -7035.965,E2 -7035.965} C_VEL
LIN {X 0,Y 481.721,Z 388.573,A -85,B 0,C 180,E1 -7036.12,E2 -7036.12} C_VEL
LIN {X 0,Y 481.712,Z 388.484,A -85,B 0,C 180,E1 -7038.722,E2 -7038.722} C_VEL
LIN {X 0,Y 481.649,Z 388.488,A -85,B 0,C 180,E1 -7041.395,E2 -7041.395} C_VEL
LIN {X 0,Y 481.674,Z 388.483,A -85,B 0,C 180,E1 -7044.113,E2 -7044.113} C_VEL
LIN {X 0,Y 481.697,Z 388.478,A -85,B 0,C 180,E1 -7047.127,E2 -7047.127} C_VEL
LIN {X 0,Y 481.676,Z 388.478,A -85,B 0,C 180,E1 -7049.741,E2 -7049.741} C_VEL
LIN {X 0,Y 481.673,Z 388.485,A -85,B 0,C 180,E1 -7052.674,E2 -7052.674} C_VEL
LIN {X 0,Y 481.637,Z 388.486,A -85,B 0,C 180,E1 -7055.71,E2 -7055.71} C_VEL
LIN {X 0,Y 481.673,Z 388.485,A -85,B 0,C 180,E1 -7058.859,E2 -7058.859} C_VEL
LIN {X 0,Y 481.649,Z 388.483,A -85,B 0,C 180,E1 -7061.912,E2 -7061.912} C_VEL
LIN {X 0,Y 481.656,Z 388.491,A -85,B 0,C 180,E1 -7064.458,E2 -7064.458} C_VEL
LIN {X 0,Y 481.645,Z 388.485,A -85,B 0,C 180,E1 -7067.839,E2 -7067.839} C_VEL
LIN {X 0,Y 481.659,Z 388.481,A -85,B 0,C 180,E1 -7070.655,E2 -7070.655} C_VEL
LIN {X 0,Y 481.62,Z 388.49,A -85,B 0,C 180,E1 -7073.458,E2 -7073.458} C_VEL
LIN {X 0,Y 481.713,Z 388.482,A -85,B 0,C 180,E1 -7076.33,E2 -7076.33} C_VEL
LIN {X 0,Y 481.67,Z 388.481,A -85,B 0,C 180,E1 -7077.098,E2 -7077.098} C_VEL
LIN {X 0,Y 480.994,Z 388.565,A -85,B 0,C 180,E1 -7077.564,E2 -7077.564} C_VEL
LIN {X 0,Y 478.14,Z 388.924,A -85,B 0,C 180,E1 -7078.291,E2 -7078.291} C_VEL
LIN {X 0,Y 475.276,Z 389.284,A -85,B 0,C 180,E1 -7079.027,E2 -7079.027} C_VEL
LIN {X 0,Y 474.602,Z 389.364,A -85,B 0,C 180,E1 -7079.502,E2 -7079.502} C_VEL
LIN {X 0,Y 474.701,Z 389.611,A -85,B 0,C 180,E1 -7080.328,E2 -7080.328} C_VEL
LIN {X 0,Y 478.469,Z 405.957,A -85,B 0,C 180,E1 -7082.696,E2 -7082.696} C_VEL
LIN {X 0,Y 478.451,Z 413,A -85,B 0,C 180,E1 -7083.642,E2 -7083.642} C_VEL
LIN {X 0,Y 477.697,Z 433.781,A -85,B 0,C 180,E1 -7086.382,E2 -7086.382} C_VEL
LIN {X 0,Y 476.99,Z 454.246,A -85,B 0,C 180,E1 -7089.065,E2 -7089.065} C_VEL
LIN {X 0,Y 476.239,Z 480.52,A -85,B 0,C 180,E1 -7092.391,E2 -7092.391} C_VEL
LIN {X 0,Y 476.066,Z 488.085,A -85,B 0,C 180,E1 -7093.286,E2 -7093.286} C_VEL
LIN {X 0,Y 478.126,Z 503.23,A -85,B 0,C 180,E1 -7093.601,E2 -7093.601} C_VEL
LIN {X 0,Y 477.393,Z 598.913,A -85,B 0,C 180,E1 -7095.071,E2 -7095.071} C_VEL
LIN {X 0,Y 477.126,Z 612.2,A -85,B 0,C 180,E1 -7095.444,E2 -7095.444} C_VEL
LIN {X 0,Y 476.699,Z 624.697,A -85,B 0,C 180,E1 -7095.975,E2 -7095.975} C_VEL
LIN {X 0,Y 476.282,Z 637.28,A -85,B 0,C 180,E1 -7096.702,E2 -7096.702} C_VEL
LIN {X 0,Y 475.89,Z 648.239,A -85,B 0,C 180,E1 -7097.527,E2 -7097.527} C_VEL
LIN {X 0,Y 475.312,Z 659.539,A -85,B 0,C 180,E1 -7098.594,E2 -7098.594} C_VEL
LIN {X 0,Y 474.937,Z 667.804,A -85,B 0,C 180,E1 -7099.556,E2 -7099.556} C_VEL
LIN {X 0,Y 474.59,Z 675.443,A -85,B 0,C 180,E1 -7100.625,E2 -7100.625} C_VEL
LIN {X 0,Y 474.249,Z 682.893,A -85,B 0,C 180,E1 -7101.907,E2 -7101.907} C_VEL
LIN {X 0,Y 474.051,Z 689.614,A -85,B 0,C 180,E1 -7103.367,E2 -7103.367} C_VEL
LIN {X 0,Y 473.849,Z 694.948,A -85,B 0,C 180,E1 -7104.895,E2 -7104.895} C_VEL
LIN {X 0,Y 473.781,Z 697.237,A -85,B 0,C 180,E1 -7105.747,E2 -7105.747} C_VEL
LIN {X 0,Y 473.808,Z 699.104,A -85,B 0,C 180,E1 -7106.599,E2 -7106.599} C_VEL
LIN {X 0,Y 473.743,Z 700.534,A -85,B 0,C 180,E1 -7107.449,E2 -7107.449} C_VEL
LIN {X 0,Y 473.688,Z 702.153,A -85,B 0,C 180,E1 -7109.15,E2 -7109.15} C_VEL
LIN {X 0,Y 473.67,Z 702.391,A -85,B 0,C 180,E1 -7110,E2 -7110} C_VEL
LIN {X 0,Y 473.688,Z 702.203,A -85,B 0,C 180,E1 -7110.85,E2 -7110.85} C_VEL
LIN {X 0,Y 473.743,Z 700.649,A -85,B 0,C 180,E1 -7112.551,E2 -7112.551} C_VEL
LIN {X 0,Y 473.808,Z 699.283,A -85,B 0,C 180,E1 -7113.402,E2 -7113.402} C_VEL
LIN {X 0,Y 473.788,Z 696.409,A -85,B 0,C 180,E1 -7114.68,E2 -7114.68} C_VEL
LIN {X 0,Y 473.939,Z 692.503,A -85,B 0,C 180,E1 -7115.958,E2 -7115.958} C_VEL
LIN {X 0,Y 474.029,Z 687.447,A -85,B 0,C 180,E1 -7117.24,E2 -7117.24} C_VEL
LIN {X 0,Y 474.331,Z 681.071,A -85,B 0,C 180,E1 -7118.521,E2 -7118.521} C_VEL
LIN {X 0,Y 474.66,Z 673.155,A -85,B 0,C 180,E1 -7119.804,E2 -7119.804} C_VEL
LIN {X 0,Y 475.037,Z 665.072,A -85,B 0,C 180,E1 -7120.873,E2 -7120.873} C_VEL
LIN {X 0,Y 475.596,Z 655.155,A -85,B 0,C 180,E1 -7121.94,E2 -7121.94} C_VEL
LIN {X 0,Y 475.941,Z 643.882,A -85,B 0,C 180,E1 -7122.916,E2 -7122.916} C_VEL
LIN {X 0,Y 476.409,Z 633.135,A -85,B 0,C 180,E1 -7123.653,E2 -7123.653} C_VEL
LIN {X 0,Y 476.881,Z 620.961,A -85,B 0,C 180,E1 -7124.292,E2 -7124.292} C_VEL
LIN {X 0,Y 477.225,Z 608.372,A -85,B 0,C 180,E1 -7124.771,E2 -7124.771} C_VEL
LIN {X 0,Y 477.492,Z 595.398,A -85,B 0,C 180,E1 -7125.09,E2 -7125.09} C_VEL
LIN {X 0,Y 478.075,Z 501.956,A -85,B 0,C 180,E1 -7126.511,E2 -7126.511} C_VEL
LIN {X 0,Y 476.055,Z 487.77,A -85,B 0,C 180,E1 -7126.823,E2 -7126.823} C_VEL
LIN {X 0,Y 476.53,Z 467.833,A -85,B 0,C 180,E1 -7129.284,E2 -7129.284} C_VEL
LIN {X 0,Y 477.387,Z 442.965,A -85,B 0,C 180,E1 -7132.505,E2 -7132.505} C_VEL
LIN {X 0,Y 478.155,Z 422.312,A -85,B 0,C 180,E1 -7135.23,E2 -7135.23} C_VEL
LIN {X 0,Y 478.549,Z 406.562,A -85,B 0,C 180,E1 -7137.307,E2 -7137.307} C_VEL
LIN {X 0,Y 474.979,Z 390.795,A -85,B 0,C 180,E1 -7139.58,E2 -7139.58} C_VEL
LIN {X 0,Y 474.641,Z 389.385,A -85,B 0,C 180,E1 -7139.86,E2 -7139.86} C_VEL
LIN {X 0,Y 474.629,Z 389.364,A -85,B 0,C 180,E1 -7143.222,E2 -7143.222} C_VEL
LIN {X 0,Y 474.577,Z 389.363,A -85,B 0,C 180,E1 -7146.325,E2 -7146.325} C_VEL
LIN {X 0,Y 474.604,Z 389.361,A -85,B 0,C 180,E1 -7149.644,E2 -7149.644} C_VEL
LIN {X 0,Y 474.572,Z 389.368,A -85,B 0,C 180,E1 -7152.94,E2 -7152.94} C_VEL
LIN {X 0,Y 474.605,Z 389.362,A -85,B 0,C 180,E1 -7155.894,E2 -7155.894} C_VEL
LIN {X 0,Y 474.604,Z 389.364,A -85,B 0,C 180,E1 -7159.045,E2 -7159.045} C_VEL
LIN {X 0,Y 474.6,Z 389.367,A -85,B 0,C 180,E1 -7161.706,E2 -7161.706} C_VEL
LIN {X 0,Y 474.62,Z 389.361,A -85,B 0,C 180,E1 -7164.725,E2 -7164.725} C_VEL
LIN {X 0,Y 474.631,Z 389.364,A -85,B 0,C 180,E1 -7167.787,E2 -7167.787} C_VEL
LIN {X 0,Y 474.601,Z 389.359,A -85,B 0,C 180,E1 -7170.891,E2 -7170.891} C_VEL
LIN {X 0,Y 474.586,Z 389.372,A -85,B 0,C 180,E1 -7173.624,E2 -7173.624} C_VEL
LIN {X 0,Y 474.638,Z 389.351,A -85,B 0,C 180,E1 -7176.642,E2 -7176.642} C_VEL
LIN {X 0,Y 474.652,Z 389.358,A -85,B 0,C 180,E1 -7180.089,E2 -7180.089} C_VEL
LIN {X 0,Y 474.6,Z 389.355,A -85,B 0,C 180,E1 -7182.772,E2 -7182.772} C_VEL
LIN {X 0,Y 474.641,Z 389.362,A -85,B 0,C 180,E1 -7185.421,E2 -7185.421} C_VEL
LIN {X 0,Y 474.696,Z 389.344,A -85,B 0,C 180,E1 -7188.037,E2 -7188.037} C_VEL
LIN {X 0,Y 474.67,Z 389.357,A -85,B 0,C 180,E1 -7191.485,E2 -7191.485} C_VEL
LIN {X 0,Y 474.741,Z 389.341,A -85,B 0,C 180,E1 -7194.052,E2 -7194.052} C_VEL
LIN {X 0,Y 474.875,Z 389.328,A -85,B 0,C 180,E1 -7197.455,E2 -7197.455} C_VEL
LIN {X 0,Y 474.883,Z 389.329,A -85,B 0,C 180,E1 -7200,E2 -7200} C_VEL
LIN {X 0,Y 474.875,Z 389.317,A -85,B 0,C 180,E1 -7202.545,E2 -7202.545} C_VEL
LIN {X 0,Y 474.739,Z 389.351,A -85,B 0,C 180,E1 -7205.948,E2 -7205.948} C_VEL
LIN {X 0,Y 474.668,Z 389.348,A -85,B 0,C 180,E1 -7208.515,E2 -7208.515} C_VEL
LIN {X 0,Y 474.697,Z 389.357,A -85,B 0,C 180,E1 -7211.963,E2 -7211.963} C_VEL
LIN {X 0,Y 474.654,Z 389.357,A -85,B 0,C 180,E1 -7215.457,E2 -7215.457} C_VEL
LIN {X 0,Y 474.591,Z 389.363,A -85,B 0,C 180,E1 -7219.013,E2 -7219.013} C_VEL
LIN {X 0,Y 474.579,Z 389.367,A -85,B 0,C 180,E1 -7221.729,E2 -7221.729} C_VEL
LIN {X 0,Y 474.624,Z 389.359,A -85,B 0,C 180,E1 -7224.495,E2 -7224.495} C_VEL
LIN {X 0,Y 474.596,Z 389.365,A -85,B 0,C 180,E1 -7227.327,E2 -7227.327} C_VEL
LIN {X 0,Y 474.597,Z 389.365,A -85,B 0,C 180,E1 -7230.231,E2 -7230.231} C_VEL
LIN {X 0,Y 474.616,Z 389.361,A -85,B 0,C 180,E1 -7233.222,E2 -7233.222} C_VEL
LIN {X 0,Y 474.572,Z 389.369,A -85,B 0,C 180,E1 -7236.325,E2 -7236.325} C_VEL
LIN {X 0,Y 474.6,Z 389.358,A -85,B 0,C 180,E1 -7239.55,E2 -7239.55} C_VEL
LIN {X 0,Y 474.567,Z 389.357,A -85,B 0,C 180,E1 -7242.94,E2 -7242.94} C_VEL
LIN {X 0,Y 474.6,Z 389.369,A -85,B 0,C 180,E1 -7245.893,E2 -7245.893} C_VEL
LIN {X 0,Y 474.582,Z 389.346,A -85,B 0,C 180,E1 -7249.047,E2 -7249.047} C_VEL
LIN {X 0,Y 474.587,Z 389.368,A -85,B 0,C 180,E1 -7251.708,E2 -7251.708} C_VEL
LIN {X 0,Y 474.603,Z 389.365,A -85,B 0,C 180,E1 -7254.723,E2 -7254.723} C_VEL
LIN {X 0,Y 474.611,Z 389.369,A -85,B 0,C 180,E1 -7257.786,E2 -7257.786} C_VEL
LIN {X 0,Y 474.634,Z 389.59,A -85,B 0,C 180,E1 -7259.629,E2 -7259.629} C_VEL
LIN {X 0,Y 478.548,Z 406.663,A -85,B 0,C 180,E1 -7262.206,E2 -7262.206} C_VEL
LIN {X 0,Y 478.158,Z 418.733,A -85,B 0,C 180,E1 -7263.836,E2 -7263.836} C_VEL
LIN {X 0,Y 477.303,Z 437.954,A -85,B 0,C 180,E1 -7266.387,E2 -7266.387} C_VEL
LIN {X 0,Y 476.489,Z 458.186,A -85,B 0,C 180,E1 -7269.042,E2 -7269.042} C_VEL
LIN {X 0,Y 475.656,Z 483.798,A -85,B 0,C 180,E1 -7272.368,E2 -7272.368} C_VEL
LIN {X 0,Y 475.469,Z 490.585,A -85,B 0,C 180,E1 -7273.22,E2 -7273.22} C_VEL
LIN {X 0,Y 477.825,Z 511.919,A -85,B 0,C 180,E1 -7273.681,E2 -7273.681} C_VEL
LIN {X 0,Y 476.912,Z 609.371,A -85,B 0,C 180,E1 -7275.301,E2 -7275.301} C_VEL
LIN {X 0,Y 476.617,Z 621.155,A -85,B 0,C 180,E1 -7275.646,E2 -7275.646} C_VEL
LIN {X 0,Y 476.276,Z 633.634,A -85,B 0,C 180,E1 -7276.18,E2 -7276.18} C_VEL
LIN {X 0,Y 475.917,Z 644.549,A -85,B 0,C 180,E1 -7276.811,E2 -7276.811} C_VEL
LIN {X 0,Y 475.522,Z 656.41,A -85,B 0,C 180,E1 -7277.698,E2 -7277.698} C_VEL
LIN {X 0,Y 475.033,Z 667.027,A -85,B 0,C 180,E1 -7278.695,E2 -7278.695} C_VEL
LIN {X 0,Y 474.65,Z 676.15,A -85,B 0,C 180,E1 -7279.765,E2 -7279.765} C_VEL
LIN {X 0,Y 474.348,Z 685.007,A -85,B 0,C 180,E1 -7281.05,E2 -7281.05} C_VEL
LIN {X 0,Y 474.087,Z 692.101,A -85,B 0,C 180,E1 -7282.333,E2 -7282.333} C_VEL
LIN {X 0,Y 473.893,Z 698.39,A -85,B 0,C 180,E1 -7283.789,E2 -7283.789} C_VEL
LIN {X 0,Y 473.889,Z 702.139,A -85,B 0,C 180,E1 -7284.895,E2 -7284.895} C_VEL
LIN {X 0,Y 473.819,Z 704.458,A -85,B 0,C 180,E1 -7285.747,E2 -7285.747} C_VEL
LIN {X 0,Y 473.875,Z 706.347,A -85,B 0,C 180,E1 -7286.599,E2 -7286.599} C_VEL
LIN {X 0,Y 473.8,Z 707.773,A -85,B 0,C 180,E1 -7287.449,E2 -7287.449} C_VEL
LIN {X 0,Y 473.78,Z 708.778,A -85,B 0,C 180,E1 -7288.3,E2 -7288.3} C_VEL
LIN {X 0,Y 473.757,Z 709.393,A -85,B 0,C 180,E1 -7289.15,E2 -7289.15} C_VEL
LIN {X 0,Y 473.76,Z 709.613,A -85,B 0,C 180,E1 -7290,E2 -7290} C_VEL
LIN {X 0,Y 473.776,Z 709.393,A -85,B 0,C 180,E1 -7290.85,E2 -7290.85} C_VEL
LIN {X 0,Y 473.808,Z 707.775,A -85,B 0,C 180,E1 -7292.55,E2 -7292.55} C_VEL
LIN {X 0,Y 473.884,Z 706.35,A -85,B 0,C 180,E1 -7293.401,E2 -7293.401} C_VEL
LIN {X 0,Y 473.847,Z 703.379,A -85,B 0,C 180,E1 -7294.679,E2 -7294.679} C_VEL
LIN {X 0,Y 473.924,Z 699.344,A -85,B 0,C 180,E1 -7295.958,E2 -7295.958} C_VEL
LIN {X 0,Y 474.044,Z 693.114,A -85,B 0,C 180,E1 -7297.454,E2 -7297.454} C_VEL
LIN {X 0,Y 474.322,Z 686.311,A -85,B 0,C 180,E1 -7298.735,E2 -7298.735} C_VEL
LIN {X 0,Y 474.538,Z 679.341,A -85,B 0,C 180,E1 -7299.806,E2 -7299.806} C_VEL
LIN {X 0,Y 474.893,Z 670.909,A -85,B 0,C 180,E1 -7300.876,E2 -7300.876} C_VEL
LIN {X 0,Y 475.33,Z 660.455,A -85,B 0,C 180,E1 -7301.946,E2 -7301.946} C_VEL
LIN {X 0,Y 475.762,Z 648.79,A -85,B 0,C 180,E1 -7302.899,E2 -7302.899} C_VEL
LIN {X 0,Y 476.162,Z 636.624,A -85,B 0,C 180,E1 -7303.66,E2 -7303.66} C_VEL
LIN {X 0,Y 476.6,Z 624.051,A -85,B 0,C 180,E1 -7304.245,E2 -7304.245} C_VEL
LIN {X 0,Y 476.846,Z 611.606,A -85,B 0,C 180,E1 -7304.647,E2 -7304.647} C_VEL
LIN {X 0,Y 477.045,Z 595.681,A -85,B 0,C 180,E1 -7304.94,E2 -7304.94} C_VEL
LIN {X 0,Y 477.473,Z 533.697,A -85,B 0,C 180,E1 -7305.903,E2 -7305.903} C_VEL
LIN {X 0,Y 477.601,Z 510.307,A -85,B 0,C 180,E1 -7306.311,E2 -7306.311} C_VEL
LIN {X 0,Y 475.245,Z 486.432,A -85,B 0,C 180,E1 -7306.844,E2 -7306.844} C_VEL
LIN {X 0,Y 475.792,Z 464.594,A -85,B 0,C 180,E1 -7309.614,E2 -7309.614} C_VEL
LIN {X 0,Y 476.458,Z 443.834,A -85,B 0,C 180,E1 -7312.323,E2 -7312.323} C_VEL
LIN {X 0,Y 477.496,Z 418.503,A -85,B 0,C 180,E1 -7315.728,E2 -7315.728} C_VEL
LIN {X 0,Y 478.023,Z 405.32,A -85,B 0,C 180,E1 -7317.563,E2 -7317.563} C_VEL
LIN {X 0,Y 475.462,Z 393.002,A -85,B 0,C 180,E1 -7319.522,E2 -7319.522} C_VEL
LIN {X 0,Y 474.604,Z 389.452,A -85,B 0,C 180,E1 -7320.169,E2 -7320.169} C_VEL
LIN {X 0,Y 474.608,Z 389.367,A -85,B 0,C 180,E1 -7323.223,E2 -7323.223} C_VEL
LIN {X 0,Y 474.568,Z 389.373,A -85,B 0,C 180,E1 -7326.326,E2 -7326.326} C_VEL
LIN {X 0,Y 474.599,Z 389.369,A -85,B 0,C 180,E1 -7329.551,E2 -7329.551} C_VEL
LIN {X 0,Y 474.569,Z 389.369,A -85,B 0,C 180,E1 -7332.94,E2 -7332.94} C_VEL
LIN {X 0,Y 474.603,Z 389.369,A -85,B 0,C 180,E1 -7335.894,E2 -7335.894} C_VEL
LIN {X 0,Y 474.592,Z 389.368,A -85,B 0,C 180,E1 -7339.339,E2 -7339.339} C_VEL
LIN {X 0,Y 474.599,Z 389.368,A -85,B 0,C 180,E1 -7341.706,E2 -7341.706} C_VEL
LIN {X 0,Y 474.621,Z 389.362,A -85,B 0,C 180,E1 -7344.725,E2 -7344.725} C_VEL
LIN {X 0,Y 474.637,Z 389.364,A -85,B 0,C 180,E1 -7347.788,E2 -7347.788} C_VEL
LIN {X 0,Y 474.609,Z 389.365,A -85,B 0,C 180,E1 -7350.888,E2 -7350.888} C_VEL
LIN {X 0,Y 474.614,Z 389.368,A -85,B 0,C 180,E1 -7353.626,E2 -7353.626} C_VEL
LIN {X 0,Y 474.637,Z 389.362,A -85,B 0,C 180,E1 -7356.642,E2 -7356.642} C_VEL
LIN {X 0,Y 474.657,Z 389.36,A -85,B 0,C 180,E1 -7360.09,E2 -7360.09} C_VEL
LIN {X 0,Y 474.65,Z 389.396,A -85,B 0,C 180,E1 -7363.439,E2 -7363.439} C_VEL
LIN {X 0,Y 474.829,Z 390.087,A -85,B 0,C 180,E1 -7363.653,E2 -7363.653} C_VEL
LIN {X 0,Y 476.311,Z 394.151,A -85,B 0,C 180,E1 -7363.835,E2 -7363.835} C_VEL
LIN {X 0,Y 478.204,Z 399.265,A -85,B 0,C 180,E1 -7364.014,E2 -7364.014} C_VEL
LIN {X 0,Y 477.392,Z 473.703,A -85,B 0,C 180,E1 -7365.343,E2 -7365.343} C_VEL
LIN {X 0,Y 477.299,Z 487.569,A -85,B 0,C 180,E1 -7365.776,E2 -7365.776} C_VEL
LIN {X 0,Y 477.164,Z 499.406,A -85,B 0,C 180,E1 -7366.315,E2 -7366.315} C_VEL
LIN {X 0,Y 476.922,Z 510.663,A -85,B 0,C 180,E1 -7366.996,E2 -7366.996} C_VEL
LIN {X 0,Y 476.594,Z 522.004,A -85,B 0,C 180,E1 -7367.87,E2 -7367.87} C_VEL
LIN {X 0,Y 476.222,Z 530.967,A -85,B 0,C 180,E1 -7368.724,E2 -7368.724} C_VEL
LIN {X 0,Y 475.93,Z 540.104,A -85,B 0,C 180,E1 -7369.793,E2 -7369.793} C_VEL
LIN {X 0,Y 475.573,Z 547.604,A -85,B 0,C 180,E1 -7370.859,E2 -7370.859} C_VEL
LIN {X 0,Y 475.261,Z 555.271,A -85,B 0,C 180,E1 -7372.212,E2 -7372.212} C_VEL
LIN {X 0,Y 475.046,Z 561.536,A -85,B 0,C 180,E1 -7373.629,E2 -7373.629} C_VEL
LIN {X 0,Y 474.753,Z 565.874,A -85,B 0,C 180,E1 -7374.904,E2 -7374.904} C_VEL
LIN {X 0,Y 474.652,Z 568.127,A -85,B 0,C 180,E1 -7375.754,E2 -7375.754} C_VEL
LIN {X 0,Y 474.694,Z 569.927,A -85,B 0,C 180,E1 -7376.605,E2 -7376.605} C_VEL
LIN {X 0,Y 474.565,Z 571.314,A -85,B 0,C 180,E1 -7377.454,E2 -7377.454} C_VEL
LIN {X 0,Y 474.554,Z 572.237,A -85,B 0,C 180,E1 -7378.303,E2 -7378.303} C_VEL
LIN {X 0,Y 474.479,Z 572.779,A -85,B 0,C 180,E1 -7379.151,E2 -7379.151} C_VEL
LIN {X 0,Y 474.448,Z 572.923,A -85,B 0,C 180,E1 -7380,E2 -7380} C_VEL
LIN {X 0,Y 474.465,Z 572.624,A -85,B 0,C 180,E1 -7380.849,E2 -7380.849} C_VEL
LIN {X 0,Y 474.393,Z 571.935,A -85,B 0,C 180,E1 -7381.698,E2 -7381.698} C_VEL
LIN {X 0,Y 474.502,Z 570.829,A -85,B 0,C 180,E1 -7382.547,E2 -7382.547} C_VEL
LIN {X 0,Y 474.444,Z 569.332,A -85,B 0,C 180,E1 -7383.397,E2 -7383.397} C_VEL
LIN {X 0,Y 474.621,Z 566.217,A -85,B 0,C 180,E1 -7384.672,E2 -7384.672} C_VEL
LIN {X 0,Y 474.738,Z 562.047,A -85,B 0,C 180,E1 -7385.948,E2 -7385.948} C_VEL
LIN {X 0,Y 475.012,Z 556.458,A -85,B 0,C 180,E1 -7387.269,E2 -7387.269} C_VEL
LIN {X 0,Y 475.225,Z 549.933,A -85,B 0,C 180,E1 -7388.505,E2 -7388.505} C_VEL
LIN {X 0,Y 475.58,Z 541.551,A -85,B 0,C 180,E1 -7389.785,E2 -7389.785} C_VEL
LIN {X 0,Y 475.782,Z 532.947,A -85,B 0,C 180,E1 -7390.856,E2 -7390.856} C_VEL
LIN {X 0,Y 476.151,Z 522.279,A -85,B 0,C 180,E1 -7391.926,E2 -7391.926} C_VEL
LIN {X 0,Y 476.554,Z 510.656,A -85,B 0,C 180,E1 -7392.857,E2 -7392.857} C_VEL
LIN {X 0,Y 476.726,Z 499.271,A -85,B 0,C 180,E1 -7393.573,E2 -7393.573} C_VEL
LIN {X 0,Y 476.967,Z 486.535,A -85,B 0,C 180,E1 -7394.18,E2 -7394.18} C_VEL
LIN {X 0,Y 477.134,Z 473.762,A -85,B 0,C 180,E1 -7394.61,E2 -7394.61} C_VEL
LIN {X 0,Y 477.208,Z 459.055,A -85,B 0,C 180,E1 -7394.908,E2 -7394.908} C_VEL
LIN {X 0,Y 477.712,Z 398.671,A -85,B 0,C 180,E1 -7395.918,E2 -7395.918} C_VEL
LIN {X 0,Y 474.858,Z 390.24,A -85,B 0,C 180,E1 -7396.176,E2 -7396.176} C_VEL
LIN {X 0,Y 474.686,Z 389.438,A -85,B 0,C 180,E1 -7396.338,E2 -7396.338} C_VEL
LIN {X 0,Y 474.666,Z 389.362,A -85,B 0,C 180,E1 -7399.01,E2 -7399.01} C_VEL
LIN {X 0,Y 474.592,Z 389.365,A -85,B 0,C 180,E1 -7401.729,E2 -7401.729} C_VEL
LIN {X 0,Y 474.653,Z 389.361,A -85,B 0,C 180,E1 -7404.493,E2 -7404.493} C_VEL
LIN {X 0,Y 474.639,Z 389.356,A -85,B 0,C 180,E1 -7407.324,E2 -7407.324} C_VEL
LIN {X 0,Y 474.606,Z 389.361,A -85,B 0,C 180,E1 -7410.23,E2 -7410.23} C_VEL
LIN {X 0,Y 474.627,Z 389.355,A -85,B 0,C 180,E1 -7413.221,E2 -7413.221} C_VEL
LIN {X 0,Y 474.59,Z 389.368,A -85,B 0,C 180,E1 -7416.324,E2 -7416.324} C_VEL
LIN {X 0,Y 474.615,Z 389.362,A -85,B 0,C 180,E1 -7419.645,E2 -7419.645} C_VEL
LIN {X 0,Y 474.602,Z 389.363,A -85,B 0,C 180,E1 -7422.233,E2 -7422.233} C_VEL
LIN {X 0,Y 474.618,Z 389.36,A -85,B 0,C 180,E1 -7425.298,E2 -7425.298} C_VEL
LIN {X 0,Y 474.617,Z 389.363,A -85,B 0,C 180,E1 -7428.214,E2 -7428.214} C_VEL
LIN {X 0,Y 474.611,Z 389.353,A -85,B 0,C 180,E1 -7431.542,E2 -7431.542} C_VEL
LIN {X 0,Y 474.624,Z 389.358,A -85,B 0,C 180,E1 -7434.726,E2 -7434.726} C_VEL
LIN {X 0,Y 474.638,Z 389.356,A -85,B 0,C 180,E1 -7437.788,E2 -7437.788} C_VEL
LIN {X 0,Y 474.602,Z 389.364,A -85,B 0,C 180,E1 -7439.502,E2 -7439.502} C_VEL
LIN {X 0,Y 474.424,Z 390.026,A -85,B 0,C 180,E1 -7439.964,E2 -7439.964} C_VEL
LIN {X 0,Y 473.846,Z 392.206,A -85,B 0,C 180,E1 -7440.494,E2 -7440.494} C_VEL
LIN {X 0,Y 472.756,Z 396.595,A -85,B 0,C 180,E1 -7441.153,E2 -7441.153} C_VEL
LIN {X 0,Y 471.674,Z 402.317,A -85,B 0,C 180,E1 -7441.86,E2 -7441.86} C_VEL
LIN {X 0,Y 471.609,Z 407.728,A -85,B 0,C 180,E1 -7442.586,E2 -7442.586} C_VEL
LIN {X 0,Y 471.62,Z 414.069,A -85,B 0,C 180,E1 -7443.445,E2 -7443.445} C_VEL
LIN {X 0,Y 470.822,Z 435.003,A -85,B 0,C 180,E1 -7446.232,E2 -7446.232} C_VEL
LIN {X 0,Y 470.075,Z 455.726,A -85,B 0,C 180,E1 -7448.972,E2 -7448.972} C_VEL
LIN {X 0,Y 469.275,Z 482.199,A -85,B 0,C 180,E1 -7452.346,E2 -7452.346} C_VEL
LIN {X 0,Y 469.138,Z 488.181,A -85,B 0,C 180,E1 -7453.035,E2 -7453.035} C_VEL
LIN {X 0,Y 471.311,Z 504.174,A -85,B 0,C 180,E1 -7453.373,E2 -7453.373} C_VEL
LIN {X 0,Y 470.55,Z 598.886,A -85,B 0,C 180,E1 -7454.848,E2 -7454.848} C_VEL
LIN {X 0,Y 470.252,Z 612.213,A -85,B 0,C 180,E1 -7455.226,E2 -7455.226} C_VEL
LIN {X 0,Y 469.828,Z 624.725,A -85,B 0,C 180,E1 -7455.766,E2 -7455.766} C_VEL
LIN {X 0,Y 469.367,Z 636.826,A -85,B 0,C 180,E1 -7456.47,E2 -7456.47} C_VEL
LIN {X 0,Y 468.95,Z 648.282,A -85,B 0,C 180,E1 -7457.339,E2 -7457.339} C_VEL
LIN {X 0,Y 468.362,Z 659.585,A -85,B 0,C 180,E1 -7458.422,E2 -7458.422} C_VEL
LIN {X 0,Y 467.938,Z 667.853,A -85,B 0,C 180,E1 -7459.398,E2 -7459.398} C_VEL
LIN {X 0,Y 467.479,Z 676.829,A -85,B 0,C 180,E1 -7460.699,E2 -7460.699} C_VEL
LIN {X 0,Y 467.163,Z 684.035,A -85,B 0,C 180,E1 -7462.001,E2 -7462.001} C_VEL
LIN {X 0,Y 466.98,Z 690.062,A -85,B 0,C 180,E1 -7463.363,E2 -7463.363} C_VEL
LIN {X 0,Y 466.791,Z 695.002,A -85,B 0,C 180,E1 -7464.817,E2 -7464.817} C_VEL
LIN {X 0,Y 466.688,Z 697.291,A -85,B 0,C 180,E1 -7465.682,E2 -7465.682} C_VEL
LIN {X 0,Y 466.706,Z 699.158,A -85,B 0,C 180,E1 -7466.547,E2 -7466.547} C_VEL
LIN {X 0,Y 466.664,Z 700.588,A -85,B 0,C 180,E1 -7467.411,E2 -7467.411} C_VEL
LIN {X 0,Y 466.59,Z 702.207,A -85,B 0,C 180,E1 -7469.137,E2 -7469.137} C_VEL
LIN {X 0,Y 466.599,Z 702.445,A -85,B 0,C 180,E1 -7470,E2 -7470} C_VEL
LIN {X 0,Y 466.59,Z 702.256,A -85,B 0,C 180,E1 -7470.863,E2 -7470.863} C_VEL
LIN {X 0,Y 466.664,Z 700.702,A -85,B 0,C 180,E1 -7472.59,E2 -7472.59} C_VEL
LIN {X 0,Y 466.706,Z 699.335,A -85,B 0,C 180,E1 -7473.453,E2 -7473.453} C_VEL
LIN {X 0,Y 466.713,Z 696.46,A -85,B 0,C 180,E1 -7474.751,E2 -7474.751} C_VEL
LIN {X 0,Y 466.855,Z 692.553,A -85,B 0,C 180,E1 -7476.049,E2 -7476.049} C_VEL
LIN {X 0,Y 466.961,Z 687.495,A -85,B 0,C 180,E1 -7477.35,E2 -7477.35} C_VEL
LIN {X 0,Y 467.292,Z 681.117,A -85,B 0,C 180,E1 -7478.65,E2 -7478.65} C_VEL
LIN {X 0,Y 467.652,Z 673.198,A -85,B 0,C 180,E1 -7479.952,E2 -7479.952} C_VEL
LIN {X 0,Y 468.058,Z 665.112,A -85,B 0,C 180,E1 -7481.037,E2 -7481.037} C_VEL
LIN {X 0,Y 468.634,Z 655.19,A -85,B 0,C 180,E1 -7482.12,E2 -7482.12} C_VEL
LIN {X 0,Y 468.989,Z 644.305,A -85,B 0,C 180,E1 -7483.079,E2 -7483.079} C_VEL
LIN {X 0,Y 469.51,Z 633.154,A -85,B 0,C 180,E1 -7483.857,E2 -7483.857} C_VEL
LIN {X 0,Y 469.987,Z 620.963,A -85,B 0,C 180,E1 -7484.506,E2 -7484.506} C_VEL
LIN {X 0,Y 470.372,Z 608.348,A -85,B 0,C 180,E1 -7484.992,E2 -7484.992} C_VEL
LIN {X 0,Y 470.638,Z 595.289,A -85,B 0,C 180,E1 -7485.315,E2 -7485.315} C_VEL
LIN {X 0,Y 471.242,Z 502.279,A -85,B 0,C 180,E1 -7486.751,E2 -7486.751} C_VEL
LIN {X 0,Y 469.114,Z 487.706,A -85,B 0,C 180,E1 -7487.082,E2 -7487.082} C_VEL
LIN {X 0,Y 469.632,Z 468.445,A -85,B 0,C 180,E1 -7489.474,E2 -7489.474} C_VEL
LIN {X 0,Y 470.485,Z 444.296,A -85,B 0,C 180,E1 -7492.63,E2 -7492.63} C_VEL
LIN {X 0,Y 471.294,Z 423.591,A -85,B 0,C 180,E1 -7495.387,E2 -7495.387} C_VEL
LIN {X 0,Y 471.76,Z 408.666,A -85,B 0,C 180,E1 -7497.373,E2 -7497.373} C_VEL
LIN {X 0,Y 468.491,Z 393.846,A -85,B 0,C 180,E1 -7499.532,E2 -7499.532} C_VEL
LIN {X 0,Y 467.614,Z 390.409,A -85,B 0,C 180,E1 -7500.076,E2 -7500.076} C_VEL
LIN {X 0,Y 467.583,Z 390.242,A -85,B 0,C 180,E1 -7502.759,E2 -7502.759} C_VEL
LIN {X 0,Y 467.548,Z 390.243,A -85,B 0,C 180,E1 -7505.891,E2 -7505.891} C_VEL
LIN {X 0,Y 467.547,Z 390.247,A -85,B 0,C 180,E1 -7509.149,E2 -7509.149} C_VEL
LIN {X 0,Y 467.561,Z 390.239,A -85,B 0,C 180,E1 -7511.405,E2 -7511.405} C_VEL
LIN {X 0,Y 467.568,Z 390.228,A -85,B 0,C 180,E1 -7515.052,E2 -7515.052} C_VEL
LIN {X 0,Y 467.565,Z 390.24,A -85,B 0,C 180,E1 -7518.726,E2 -7518.726} C_VEL
LIN {X 0,Y 467.549,Z 390.241,A -85,B 0,C 180,E1 -7521.954,E2 -7521.954} C_VEL
LIN {X 0,Y 467.557,Z 390.243,A -85,B 0,C 180,E1 -7525.167,E2 -7525.167} C_VEL
LIN {X 0,Y 467.581,Z 390.24,A -85,B 0,C 180,E1 -7528.26,E2 -7528.26} C_VEL
LIN {X 0,Y 467.547,Z 390.24,A -85,B 0,C 180,E1 -7531.248,E2 -7531.248} C_VEL
LIN {X 0,Y 467.58,Z 390.238,A -85,B 0,C 180,E1 -7534.401,E2 -7534.401} C_VEL
LIN {X 0,Y 467.58,Z 390.231,A -85,B 0,C 180,E1 -7536.996,E2 -7536.996} C_VEL
LIN {X 0,Y 467.623,Z 390.238,A -85,B 0,C 180,E1 -7539.777,E2 -7539.777} C_VEL
LIN {X 0,Y 467.572,Z 390.231,A -85,B 0,C 180,E1 -7542.505,E2 -7542.505} C_VEL
LIN {X 0,Y 467.599,Z 390.237,A -85,B 0,C 180,E1 -7545.196,E2 -7545.196} C_VEL
LIN {X 0,Y 467.652,Z 390.223,A -85,B 0,C 180,E1 -7547.854,E2 -7547.854} C_VEL
LIN {X 0,Y 467.638,Z 390.231,A -85,B 0,C 180,E1 -7551.356,E2 -7551.356} C_VEL
LIN {X 0,Y 467.706,Z 390.218,A -85,B 0,C 180,E1 -7553.962,E2 -7553.962} C_VEL
LIN {X 0,Y 467.815,Z 390.206,A -85,B 0,C 180,E1 -7557.417,E2 -7557.417} C_VEL
LIN {X 0,Y 467.853,Z 390.205,A -85,B 0,C 180,E1 -7560,E2 -7560} C_VEL
LIN {X 0,Y 467.815,Z 390.196,A -85,B 0,C 180,E1 -7562.583,E2 -7562.583} C_VEL
LIN {X 0,Y 467.704,Z 390.226,A -85,B 0,C 180,E1 -7566.038,E2 -7566.038} C_VEL
LIN {X 0,Y 467.637,Z 390.223,A -85,B 0,C 180,E1 -7568.644,E2 -7568.644} C_VEL
LIN {X 0,Y 467.652,Z 390.23,A -85,B 0,C 180,E1 -7572.354,E2 -7572.354} C_VEL
LIN {X 0,Y 467.574,Z 390.233,A -85,B 0,C 180,E1 -7575.85,E2 -7575.85} C_VEL
LIN {X 0,Y 467.571,Z 390.237,A -85,B 0,C 180,E1 -7578.746,E2 -7578.746} C_VEL
LIN {X 0,Y 467.526,Z 390.239,A -85,B 0,C 180,E1 -7582.074,E2 -7582.074} C_VEL
LIN {X 0,Y 467.553,Z 390.239,A -85,B 0,C 180,E1 -7584.89,E2 -7584.89} C_VEL
LIN {X 0,Y 467.545,Z 390.243,A -85,B 0,C 180,E1 -7587.774,E2 -7587.774} C_VEL
LIN {X 0,Y 467.548,Z 390.241,A -85,B 0,C 180,E1 -7591.04,E2 -7591.04} C_VEL
LIN {X 0,Y 467.578,Z 390.234,A -85,B 0,C 180,E1 -7594.239,E2 -7594.239} C_VEL
LIN {X 0,Y 467.516,Z 390.247,A -85,B 0,C 180,E1 -7597.18,E2 -7597.18} C_VEL
LIN {X 0,Y 467.519,Z 390.226,A -85,B 0,C 180,E1 -7600.271,E2 -7600.271} C_VEL
LIN {X 0,Y 467.518,Z 390.235,A -85,B 0,C 180,E1 -7602.568,E2 -7602.568} C_VEL
LIN {X 0,Y 467.564,Z 390.24,A -85,B 0,C 180,E1 -7605.052,E2 -7605.052} C_VEL
LIN {X 0,Y 467.552,Z 390.22,A -85,B 0,C 180,E1 -7608.727,E2 -7608.727} C_VEL
LIN {X 0,Y 467.538,Z 390.25,A -85,B 0,C 180,E1 -7611.952,E2 -7611.952} C_VEL
LIN {X 0,Y 467.54,Z 390.245,A -85,B 0,C 180,E1 -7615.165,E2 -7615.165} C_VEL
LIN {X 0,Y 467.544,Z 390.249,A -85,B 0,C 180,E1 -7618.257,E2 -7618.257} C_VEL
LIN {X 0,Y 467.595,Z 390.474,A -85,B 0,C 180,E1 -7619.377,E2 -7619.377} C_VEL
LIN {X 0,Y 471.607,Z 407.875,A -85,B 0,C 180,E1 -7622.053,E2 -7622.053} C_VEL
LIN {X 0,Y 471.55,Z 414.456,A -85,B 0,C 180,E1 -7622.962,E2 -7622.962} C_VEL
LIN {X 0,Y 470.465,Z 436.434,A -85,B 0,C 180,E1 -7625.93,E2 -7625.93} C_VEL
LIN {X 0,Y 469.486,Z 459.032,A -85,B 0,C 180,E1 -7628.944,E2 -7628.944} C_VEL
LIN {X 0,Y 468.622,Z 484.638,A -85,B 0,C 180,E1 -7632.32,E2 -7632.32} C_VEL
LIN {X 0,Y 468.471,Z 489.612,A -85,B 0,C 180,E1 -7632.957,E2 -7632.957} C_VEL
LIN {X 0,Y 469.44,Z 498.629,A -85,B 0,C 180,E1 -7633.178,E2 -7633.178} C_VEL
LIN {X 0,Y 470.946,Z 514.098,A -85,B 0,C 180,E1 -7633.498,E2 -7633.498} C_VEL
LIN {X 0,Y 470.284,Z 586.832,A -85,B 0,C 180,E1 -7634.701,E2 -7634.701} C_VEL
LIN {X 0,Y 470.058,Z 609.414,A -85,B 0,C 180,E1 -7635.081,E2 -7635.081} C_VEL
LIN {X 0,Y 469.752,Z 621.16,A -85,B 0,C 180,E1 -7635.432,E2 -7635.432} C_VEL
LIN {X 0,Y 469.385,Z 633.619,A -85,B 0,C 180,E1 -7635.973,E2 -7635.973} C_VEL
LIN {X 0,Y 468.954,Z 645.467,A -85,B 0,C 180,E1 -7636.678,E2 -7636.678} C_VEL
LIN {X 0,Y 468.56,Z 656.68,A -85,B 0,C 180,E1 -7637.538,E2 -7637.538} C_VEL
LIN {X 0,Y 468.06,Z 666.987,A -85,B 0,C 180,E1 -7638.524,E2 -7638.524} C_VEL
LIN {X 0,Y 467.638,Z 676.106,A -85,B 0,C 180,E1 -7639.61,E2 -7639.61} C_VEL
LIN {X 0,Y 467.287,Z 684.96,A -85,B 0,C 180,E1 -7640.914,E2 -7640.914} C_VEL
LIN {X 0,Y 467.032,Z 692.052,A -85,B 0,C 180,E1 -7642.216,E2 -7642.216} C_VEL
LIN {X 0,Y 466.864,Z 697.563,A -85,B 0,C 180,E1 -7643.485,E2 -7643.485} C_VEL
LIN {X 0,Y 466.821,Z 702.088,A -85,B 0,C 180,E1 -7644.817,E2 -7644.817} C_VEL
LIN {X 0,Y 466.724,Z 704.405,A -85,B 0,C 180,E1 -7645.682,E2 -7645.682} C_VEL
LIN {X 0,Y 466.782,Z 706.294,A -85,B 0,C 180,E1 -7646.547,E2 -7646.547} C_VEL
LIN {X 0,Y 466.719,Z 707.72,A -85,B 0,C 180,E1 -7647.411,E2 -7647.411} C_VEL
LIN {X 0,Y 466.683,Z 709.339,A -85,B 0,C 180,E1 -7649.137,E2 -7649.137} C_VEL
LIN {X 0,Y 466.684,Z 709.56,A -85,B 0,C 180,E1 -7650,E2 -7650} C_VEL
LIN {X 0,Y 466.702,Z 709.339,A -85,B 0,C 180,E1 -7650.863,E2 -7650.863} C_VEL
LIN {X 0,Y 466.726,Z 707.721,A -85,B 0,C 180,E1 -7652.589,E2 -7652.589} C_VEL
LIN {X 0,Y 466.791,Z 706.296,A -85,B 0,C 180,E1 -7653.453,E2 -7653.453} C_VEL
LIN {X 0,Y 466.77,Z 703.327,A -85,B 0,C 180,E1 -7654.75,E2 -7654.75} C_VEL
LIN {X 0,Y 466.828,Z 699.292,A -85,B 0,C 180,E1 -7656.049,E2 -7656.049} C_VEL
LIN {X 0,Y 466.993,Z 693.063,A -85,B 0,C 180,E1 -7657.567,E2 -7657.567} C_VEL
LIN {X 0,Y 467.28,Z 686.262,A -85,B 0,C 180,E1 -7658.868,E2 -7658.868} C_VEL
LIN {X 0,Y 467.534,Z 679.293,A -85,B 0,C 180,E1 -7659.955,E2 -7659.955} C_VEL
LIN {X 0,Y 467.88,Z 670.863,A -85,B 0,C 180,E1 -7661.041,E2 -7661.041} C_VEL
LIN {X 0,Y 468.362,Z 660.414,A -85,B 0,C 180,E1 -7662.127,E2 -7662.127} C_VEL
LIN {X 0,Y 468.781,Z 650.041,A -85,B 0,C 180,E1 -7662.996,E2 -7662.996} C_VEL
LIN {X 0,Y 469.188,Z 638.572,A -85,B 0,C 180,E1 -7663.756,E2 -7663.756} C_VEL
LIN {X 0,Y 469.63,Z 626.618,A -85,B 0,C 180,E1 -7664.351,E2 -7664.351} C_VEL
LIN {X 0,Y 469.957,Z 613.626,A -85,B 0,C 180,E1 -7664.811,E2 -7664.811} C_VEL
LIN {X 0,Y 470.133,Z 601.119,A -85,B 0,C 180,E1 -7665.082,E2 -7665.082} C_VEL
LIN {X 0,Y 470.651,Z 532.021,A -85,B 0,C 180,E1 -7666.161,E2 -7666.161} C_VEL
LIN {X 0,Y 470.784,Z 511.048,A -85,B 0,C 180,E1 -7666.539,E2 -7666.539} C_VEL
LIN {X 0,Y 468.256,Z 485.038,A -85,B 0,C 180,E1 -7667.143,E2 -7667.143} C_VEL
LIN {X 0,Y 468.867,Z 461.749,A -85,B 0,C 180,E1 -7670.167,E2 -7670.167} C_VEL
LIN {X 0,Y 469.708,Z 439.64,A -85,B 0,C 180,E1 -7673.127,E2 -7673.127} C_VEL
LIN {X 0,Y 470.64,Z 418.477,A -85,B 0,C 180,E1 -7676.048,E2 -7676.048} C_VEL
LIN {X 0,Y 471.238,Z 407.986,A -85,B 0,C 180,E1 -7677.538,E2 -7677.538} C_VEL
LIN {X 0,Y 469.787,Z 399.783,A -85,B 0,C 180,E1 -7678.843,E2 -7678.843} C_VEL
LIN {X 0,Y 467.539,Z 390.367,A -85,B 0,C 180,E1 -7680.486,E2 -7680.486} C_VEL
LIN {X 0,Y 467.552,Z 390.248,A -85,B 0,C 180,E1 -7683.791,E2 -7683.791} C_VEL
LIN {X 0,Y 467.503,Z 390.251,A -85,B 0,C 180,E1 -7686.965,E2 -7686.965} C_VEL
LIN {X 0,Y 467.544,Z 390.249,A -85,B 0,C 180,E1 -7689.949,E2 -7689.949} C_VEL
LIN {X 0,Y 467.517,Z 390.248,A -85,B 0,C 180,E1 -7692.568,E2 -7692.568} C_VEL
LIN {X 0,Y 467.566,Z 390.242,A -85,B 0,C 180,E1 -7695.052,E2 -7695.052} C_VEL
LIN {X 0,Y 467.561,Z 390.241,A -85,B 0,C 180,E1 -7698.726,E2 -7698.726} C_VEL
LIN {X 0,Y 467.548,Z 390.245,A -85,B 0,C 180,E1 -7701.954,E2 -7701.954} C_VEL
LIN {X 0,Y 467.558,Z 390.245,A -85,B 0,C 180,E1 -7705.167,E2 -7705.167} C_VEL
LIN {X 0,Y 467.585,Z 390.24,A -85,B 0,C 180,E1 -7708.26,E2 -7708.26} C_VEL
LIN {X 0,Y 467.557,Z 390.244,A -85,B 0,C 180,E1 -7711.249,E2 -7711.249} C_VEL
LIN {X 0,Y 467.584,Z 390.239,A -85,B 0,C 180,E1 -7714.158,E2 -7714.158} C_VEL
LIN {X 0,Y 467.578,Z 390.243,A -85,B 0,C 180,E1 -7716.996,E2 -7716.996} C_VEL
LIN {X 0,Y 467.625,Z 390.238,A -85,B 0,C 180,E1 -7719.777,E2 -7719.777} C_VEL
LIN {X 0,Y 467.593,Z 390.243,A -85,B 0,C 180,E1 -7722.957,E2 -7722.957} C_VEL
LIN {X 0,Y 467.648,Z 390.582,A -85,B 0,C 180,E1 -7723.297,E2 -7723.297} C_VEL
LIN {X 0,Y 467.846,Z 391.395,A -85,B 0,C 180,E1 -7723.392,E2 -7723.392} C_VEL
LIN {X 0,Y 471.499,Z 400.932,A -85,B 0,C 180,E1 -7723.754,E2 -7723.754} C_VEL
LIN {X 0,Y 470.578,Z 475.019,A -85,B 0,C 180,E1 -7725.126,E2 -7725.126} C_VEL
LIN {X 0,Y 470.53,Z 488.807,A -85,B 0,C 180,E1 -7725.567,E2 -7725.567} C_VEL
LIN {X 0,Y 470.367,Z 500.622,A -85,B 0,C 180,E1 -7726.114,E2 -7726.114} C_VEL
LIN {X 0,Y 470.097,Z 511.871,A -85,B 0,C 180,E1 -7726.804,E2 -7726.804} C_VEL
LIN {X 0,Y 469.748,Z 523.209,A -85,B 0,C 180,E1 -7727.69,E2 -7727.69} C_VEL
LIN {X 0,Y 469.362,Z 532.169,A -85,B 0,C 180,E1 -7728.557,E2 -7728.557} C_VEL
LIN {X 0,Y 469.055,Z 541.297,A -85,B 0,C 180,E1 -7729.642,E2 -7729.642} C_VEL
LIN {X 0,Y 468.668,Z 548.767,A -85,B 0,C 180,E1 -7730.723,E2 -7730.723} C_VEL
LIN {X 0,Y 468.359,Z 556.129,A -85,B 0,C 180,E1 -7732.043,E2 -7732.043} C_VEL
LIN {X 0,Y 468.173,Z 560.914,A -85,B 0,C 180,E1 -7733.103,E2 -7733.103} C_VEL
LIN {X 0,Y 467.931,Z 565.618,A -85,B 0,C 180,E1 -7734.398,E2 -7734.398} C_VEL
LIN {X 0,Y 467.656,Z 569.21,A -85,B 0,C 180,E1 -7735.691,E2 -7735.691} C_VEL
LIN {X 0,Y 467.688,Z 571.005,A -85,B 0,C 180,E1 -7736.554,E2 -7736.554} C_VEL
LIN {X 0,Y 467.576,Z 572.376,A -85,B 0,C 180,E1 -7737.416,E2 -7737.416} C_VEL
LIN {X 0,Y 467.541,Z 573.291,A -85,B 0,C 180,E1 -7738.277,E2 -7738.277} C_VEL
LIN {X 0,Y 467.46,Z 573.82,A -85,B 0,C 180,E1 -7739.139,E2 -7739.139} C_VEL
LIN {X 0,Y 467.428,Z 573.948,A -85,B 0,C 180,E1 -7740,E2 -7740} C_VEL
LIN {X 0,Y 467.445,Z 573.628,A -85,B 0,C 180,E1 -7740.862,E2 -7740.862} C_VEL
LIN {X 0,Y 467.37,Z 572.919,A -85,B 0,C 180,E1 -7741.723,E2 -7741.723} C_VEL
LIN {X 0,Y 467.483,Z 571.789,A -85,B 0,C 180,E1 -7742.585,E2 -7742.585} C_VEL
LIN {X 0,Y 467.476,Z 569.312,A -85,B 0,C 180,E1 -7743.879,E2 -7743.879} C_VEL
LIN {X 0,Y 467.58,Z 565.817,A -85,B 0,C 180,E1 -7745.174,E2 -7745.174} C_VEL
LIN {X 0,Y 467.829,Z 561.207,A -85,B 0,C 180,E1 -7746.469,E2 -7746.469} C_VEL
LIN {X 0,Y 468.097,Z 555.361,A -85,B 0,C 180,E1 -7747.766,E2 -7747.766} C_VEL
LIN {X 0,Y 468.342,Z 548.026,A -85,B 0,C 180,E1 -7749.066,E2 -7749.066} C_VEL
LIN {X 0,Y 468.663,Z 538.891,A -85,B 0,C 180,E1 -7750.367,E2 -7750.367} C_VEL
LIN {X 0,Y 469.021,Z 529.45,A -85,B 0,C 180,E1 -7751.452,E2 -7751.452} C_VEL
LIN {X 0,Y 469.348,Z 520.224,A -85,B 0,C 180,E1 -7752.321,E2 -7752.321} C_VEL
LIN {X 0,Y 469.659,Z 508.171,A -85,B 0,C 180,E1 -7753.236,E2 -7753.236} C_VEL
LIN {X 0,Y 469.882,Z 495.952,A -85,B 0,C 180,E1 -7753.956,E2 -7753.956} C_VEL
LIN {X 0,Y 470.156,Z 482.608,A -85,B 0,C 180,E1 -7754.528,E2 -7754.528} C_VEL
LIN {X 0,Y 470.238,Z 469.428,A -85,B 0,C 180,E1 -7754.913,E2 -7754.913} C_VEL
LIN {X 0,Y 470.853,Z 400.218,A -85,B 0,C 180,E1 -7756.108,E2 -7756.108} C_VEL
LIN {X 0,Y 467.764,Z 390.996,A -85,B 0,C 180,E1 -7756.403,E2 -7756.403} C_VEL
LIN {X 0,Y 467.62,Z 390.288,A -85,B 0,C 180,E1 -7756.592,E2 -7756.592} C_VEL
LIN {X 0,Y 467.625,Z 390.237,A -85,B 0,C 180,E1 -7759.308,E2 -7759.308} C_VEL
LIN {X 0,Y 467.538,Z 390.245,A -85,B 0,C 180,E1 -7762.074,E2 -7762.074} C_VEL
LIN {X 0,Y 467.595,Z 390.243,A -85,B 0,C 180,E1 -7764.888,E2 -7764.888} C_VEL
LIN {X 0,Y 467.582,Z 390.233,A -85,B 0,C 180,E1 -7767.772,E2 -7767.772} C_VEL
LIN {X 0,Y 467.571,Z 390.243,A -85,B 0,C 180,E1 -7771.045,E2 -7771.045} C_VEL
LIN {X 0,Y 467.579,Z 390.233,A -85,B 0,C 180,E1 -7774.24,E2 -7774.24} C_VEL
LIN {X 0,Y 467.549,Z 390.24,A -85,B 0,C 180,E1 -7777.186,E2 -7777.186} C_VEL
LIN {X 0,Y 467.574,Z 390.242,A -85,B 0,C 180,E1 -7780.265,E2 -7780.265} C_VEL
LIN {X 0,Y 467.55,Z 390.243,A -85,B 0,C 180,E1 -7783.745,E2 -7783.745} C_VEL
LIN {X 0,Y 467.551,Z 390.243,A -85,B 0,C 180,E1 -7786.255,E2 -7786.255} C_VEL
LIN {X 0,Y 467.572,Z 390.24,A -85,B 0,C 180,E1 -7789.735,E2 -7789.735} C_VEL
LIN {X 0,Y 467.545,Z 390.246,A -85,B 0,C 180,E1 -7792.815,E2 -7792.815} C_VEL
LIN {X 0,Y 467.589,Z 390.24,A -85,B 0,C 180,E1 -7796.212,E2 -7796.212} C_VEL
LIN {X 0,Y 467.566,Z 390.24,A -85,B 0,C 180,E1 -7799.502,E2 -7799.502} C_VEL
LIN {X 0,Y 467.656,Z 390.485,A -85,B 0,C 180,E1 -7800.052,E2 -7800.052} C_VEL
LIN {X 0,Y 471.501,Z 406.983,A -85,B 0,C 180,E1 -7802.479,E2 -7802.479} C_VEL
LIN {X 0,Y 471.609,Z 407.728,A -85,B 0,C 180,E1 -7802.586,E2 -7802.586} C_VEL
LIN {X 0,Y 471.584,Z 410.341,A -85,B 0,C 180,E1 -7802.939,E2 -7802.939} C_VEL
LIN {X 0,Y 470.928,Z 413.058,A -85,B 0,C 180,E1 -7803.273,E2 -7803.273} C_VEL
LIN {X 0,Y 468.513,Z 418.587,A -85,B 0,C 180,E1 -7803.901,E2 -7803.901} C_VEL
LIN {X 0,Y 465.241,Z 425.586,A -85,B 0,C 180,E1 -7804.692,E2 -7804.692} C_VEL
LIN {X 0,Y 464.279,Z 429.737,A -85,B 0,C 180,E1 -7805.211,E2 -7805.211} C_VEL
LIN {X 0,Y 463.273,Z 453.722,A -85,B 0,C 180,E1 -7808.415,E2 -7808.415} C_VEL
LIN {X 0,Y 462.486,Z 476.662,A -85,B 0,C 180,E1 -7811.39,E2 -7811.39} C_VEL
LIN {X 0,Y 462.247,Z 487.742,A -85,B 0,C 180,E1 -7812.753,E2 -7812.753} C_VEL
LIN {X 0,Y 464.508,Z 504.137,A -85,B 0,C 180,E1 -7813.122,E2 -7813.122} C_VEL
LIN {X 0,Y 463.708,Z 598.863,A -85,B 0,C 180,E1 -7814.619,E2 -7814.619} C_VEL
LIN {X 0,Y 463.401,Z 612.228,A -85,B 0,C 180,E1 -7815.003,E2 -7815.003} C_VEL
LIN {X 0,Y 462.947,Z 624.755,A -85,B 0,C 180,E1 -7815.55,E2 -7815.55} C_VEL
LIN {X 0,Y 462.47,Z 636.863,A -85,B 0,C 180,E1 -7816.264,E2 -7816.264} C_VEL
LIN {X 0,Y 462.064,Z 647.258,A -85,B 0,C 180,E1 -7817.052,E2 -7817.052} C_VEL
LIN {X 0,Y 461.529,Z 657.563,A -85,B 0,C 180,E1 -7818.026,E2 -7818.026} C_VEL
LIN {X 0,Y 460.937,Z 667.902,A -85,B 0,C 180,E1 -7819.235,E2 -7819.235} C_VEL
LIN {X 0,Y 460.459,Z 676.88,A -85,B 0,C 180,E1 -7820.556,E2 -7820.556} C_VEL
LIN {X 0,Y 460.103,Z 684.088,A -85,B 0,C 180,E1 -7821.877,E2 -7821.877} C_VEL
LIN {X 0,Y 459.89,Z 690.561,A -85,B 0,C 180,E1 -7823.378,E2 -7823.378} C_VEL
LIN {X 0,Y 459.733,Z 695.055,A -85,B 0,C 180,E1 -7824.737,E2 -7824.737} C_VEL
LIN {X 0,Y 459.602,Z 697.345,A -85,B 0,C 180,E1 -7825.615,E2 -7825.615} C_VEL
LIN {X 0,Y 459.604,Z 699.212,A -85,B 0,C 180,E1 -7826.493,E2 -7826.493} C_VEL
LIN {X 0,Y 459.587,Z 700.642,A -85,B 0,C 180,E1 -7827.371,E2 -7827.371} C_VEL
LIN {X 0,Y 459.495,Z 702.262,A -85,B 0,C 180,E1 -7829.124,E2 -7829.124} C_VEL
LIN {X 0,Y 459.501,Z 702.499,A -85,B 0,C 180,E1 -7830,E2 -7830} C_VEL
LIN {X 0,Y 459.495,Z 702.31,A -85,B 0,C 180,E1 -7830.877,E2 -7830.877} C_VEL
LIN {X 0,Y 459.587,Z 700.754,A -85,B 0,C 180,E1 -7832.63,E2 -7832.63} C_VEL
LIN {X 0,Y 459.604,Z 699.388,A -85,B 0,C 180,E1 -7833.507,E2 -7833.507} C_VEL
LIN {X 0,Y 459.643,Z 696.511,A -85,B 0,C 180,E1 -7834.824,E2 -7834.824} C_VEL
LIN {X 0,Y 459.767,Z 692.604,A -85,B 0,C 180,E1 -7836.143,E2 -7836.143} C_VEL
LIN {X 0,Y 459.921,Z 687.543,A -85,B 0,C 180,E1 -7837.463,E2 -7837.463} C_VEL
LIN {X 0,Y 460.24,Z 681.164,A -85,B 0,C 180,E1 -7838.784,E2 -7838.784} C_VEL
LIN {X 0,Y 460.652,Z 673.242,A -85,B 0,C 180,E1 -7840.105,E2 -7840.105} C_VEL
LIN {X 0,Y 461.072,Z 665.153,A -85,B 0,C 180,E1 -7841.207,E2 -7841.207} C_VEL
LIN {X 0,Y 461.688,Z 655.226,A -85,B 0,C 180,E1 -7842.305,E2 -7842.305} C_VEL
LIN {X 0,Y 462.036,Z 645.082,A -85,B 0,C 180,E1 -7843.219,E2 -7843.219} C_VEL
LIN {X 0,Y 462.618,Z 633.176,A -85,B 0,C 180,E1 -7844.068,E2 -7844.068} C_VEL
LIN {X 0,Y 463.127,Z 620.968,A -85,B 0,C 180,E1 -7844.725,E2 -7844.725} C_VEL
LIN {X 0,Y 463.522,Z 608.329,A -85,B 0,C 180,E1 -7845.218,E2 -7845.218} C_VEL
LIN {X 0,Y 463.807,Z 595.189,A -85,B 0,C 180,E1 -7845.546,E2 -7845.546} C_VEL
LIN {X 0,Y 464.425,Z 502.828,A -85,B 0,C 180,E1 -7846.994,E2 -7846.994} C_VEL
LIN {X 0,Y 462.235,Z 487.676,A -85,B 0,C 180,E1 -7847.344,E2 -7847.344} C_VEL
LIN {X 0,Y 462.806,Z 467.079,A -85,B 0,C 180,E1 -7849.933,E2 -7849.933} C_VEL
LIN {X 0,Y 463.747,Z 442.318,A -85,B 0,C 180,E1 -7853.205,E2 -7853.205} C_VEL
LIN {X 0,Y 464.529,Z 423.126,A -85,B 0,C 180,E1 -7855.784,E2 -7855.784} C_VEL
LIN {X 0,Y 464.989,Z 410.711,A -85,B 0,C 180,E1 -7857.451,E2 -7857.451} C_VEL
LIN {X 0,Y 461.889,Z 396.47,A -85,B 0,C 180,E1 -7859.549,E2 -7859.549} C_VEL
LIN {X 0,Y 460.555,Z 391.282,A -85,B 0,C 180,E1 -7860.364,E2 -7860.364} C_VEL
LIN {X 0,Y 460.523,Z 391.12,A -85,B 0,C 180,E1 -7863.326,E2 -7863.326} C_VEL
LIN {X 0,Y 460.464,Z 391.12,A -85,B 0,C 180,E1 -7866.531,E2 -7866.531} C_VEL
LIN {X 0,Y 460.513,Z 391.113,A -85,B 0,C 180,E1 -7869.865,E2 -7869.865} C_VEL
LIN {X 0,Y 460.465,Z 391.126,A -85,B 0,C 180,E1 -7872.894,E2 -7872.894} C_VEL
LIN {X 0,Y 460.507,Z 391.115,A -85,B 0,C 180,E1 -7875.832,E2 -7875.832} C_VEL
LIN {X 0,Y 460.519,Z 391.118,A -85,B 0,C 180,E1 -7878.987,E2 -7878.987} C_VEL
LIN {X 0,Y 460.49,Z 391.117,A -85,B 0,C 180,E1 -7882.376,E2 -7882.376} C_VEL
LIN {X 0,Y 460.538,Z 391.118,A -85,B 0,C 180,E1 -7885.623,E2 -7885.623} C_VEL
LIN {X 0,Y 460.541,Z 391.115,A -85,B 0,C 180,E1 -7888.745,E2 -7888.745} C_VEL
LIN {X 0,Y 460.51,Z 391.119,A -85,B 0,C 180,E1 -7891.764,E2 -7891.764} C_VEL
LIN {X 0,Y 460.524,Z 391.116,A -85,B 0,C 180,E1 -7894.703,E2 -7894.703} C_VEL
LIN {X 0,Y 460.514,Z 391.116,A -85,B 0,C 180,E1 -7897.571,E2 -7897.571} C_VEL
LIN {X 0,Y 460.569,Z 391.109,A -85,B 0,C 180,E1 -7900.384,E2 -7900.384} C_VEL
LIN {X 0,Y 460.57,Z 391.114,A -85,B 0,C 180,E1 -7904.058,E2 -7904.058} C_VEL
LIN {X 0,Y 460.607,Z 391.103,A -85,B 0,C 180,E1 -7907.666,E2 -7907.666} C_VEL
LIN {X 0,Y 460.593,Z 391.108,A -85,B 0,C 180,E1 -7911.223,E2 -7911.223} C_VEL
LIN {X 0,Y 460.672,Z 391.095,A -85,B 0,C 180,E1 -7913.87,E2 -7913.87} C_VEL
LIN {X 0,Y 460.759,Z 391.085,A -85,B 0,C 180,E1 -7917.377,E2 -7917.377} C_VEL
LIN {X 0,Y 460.822,Z 391.08,A -85,B 0,C 180,E1 -7920,E2 -7920} C_VEL
LIN {X 0,Y 460.759,Z 391.075,A -85,B 0,C 180,E1 -7922.623,E2 -7922.623} C_VEL
LIN {X 0,Y 460.671,Z 391.101,A -85,B 0,C 180,E1 -7926.13,E2 -7926.13} C_VEL
LIN {X 0,Y 460.591,Z 391.1,A -85,B 0,C 180,E1 -7928.777,E2 -7928.777} C_VEL
LIN {X 0,Y 460.601,Z 391.107,A -85,B 0,C 180,E1 -7932.435,E2 -7932.435} C_VEL
LIN {X 0,Y 460.529,Z 391.109,A -85,B 0,C 180,E1 -7935.964,E2 -7935.964} C_VEL
LIN {X 0,Y 460.528,Z 391.114,A -85,B 0,C 180,E1 -7938.884,E2 -7938.884} C_VEL
LIN {X 0,Y 460.506,Z 391.11,A -85,B 0,C 180,E1 -7942.429,E2 -7942.429} C_VEL
LIN {X 0,Y 460.513,Z 391.117,A -85,B 0,C 180,E1 -7945.297,E2 -7945.297} C_VEL
LIN {X 0,Y 460.508,Z 391.113,A -85,B 0,C 180,E1 -7948.236,E2 -7948.236} C_VEL
LIN {X 0,Y 460.523,Z 391.117,A -85,B 0,C 180,E1 -7951.282,E2 -7951.282} C_VEL
LIN {X 0,Y 460.522,Z 391.112,A -85,B 0,C 180,E1 -7954.503,E2 -7954.503} C_VEL
LIN {X 0,Y 460.483,Z 391.127,A -85,B 0,C 180,E1 -7957.625,E2 -7957.625} C_VEL
LIN {X 0,Y 460.501,Z 391.097,A -85,B 0,C 180,E1 -7961.015,E2 -7961.015} C_VEL
LIN {X 0,Y 460.508,Z 391.119,A -85,B 0,C 180,E1 -7964.59,E2 -7964.59} C_VEL
LIN {X 0,Y 460.472,Z 391.112,A -85,B 0,C 180,E1 -7967.812,E2 -7967.812} C_VEL
LIN {X 0,Y 460.477,Z 391.114,A -85,B 0,C 180,E1 -7970.131,E2 -7970.131} C_VEL
LIN {X 0,Y 460.458,Z 391.129,A -85,B 0,C 180,E1 -7973.468,E2 -7973.468} C_VEL
LIN {X 0,Y 460.502,Z 391.123,A -85,B 0,C 180,E1 -7976.673,E2 -7976.673} C_VEL
LIN {X 0,Y 460.516,Z 391.318,A -85,B 0,C 180,E1 -7979.125,E2 -7979.125} C_VEL
LIN {X 0,Y 464.579,Z 408.731,A -85,B 0,C 180,E1 -7981.844,E2 -7981.844} C_VEL
LIN {X 0,Y 464.76,Z 413.558,A -85,B 0,C 180,E1 -7982.534,E2 -7982.534} C_VEL
LIN {X 0,Y 463.618,Z 435.59,A -85,B 0,C 180,E1 -7985.557,E2 -7985.557} C_VEL
LIN {X 0,Y 462.562,Z 458.147,A -85,B 0,C 180,E1 -7988.614,E2 -7988.614} C_VEL
LIN {X 0,Y 461.679,Z 482.042,A -85,B 0,C 180,E1 -7991.816,E2 -7991.816} C_VEL
LIN {X 0,Y 461.454,Z 489.03,A -85,B 0,C 180,E1 -7992.722,E2 -7992.722} C_VEL
LIN {X 0,Y 464.096,Z 514.168,A -85,B 0,C 180,E1 -7993.278,E2 -7993.278} C_VEL
LIN {X 0,Y 463.594,Z 564.212,A -85,B 0,C 180,E1 -7994.118,E2 -7994.118} C_VEL
LIN {X 0,Y 463.224,Z 608.332,A -85,B 0,C 180,E1 -7994.828,E2 -7994.828} C_VEL
LIN {X 0,Y 462.915,Z 620.41,A -85,B 0,C 180,E1 -7995.183,E2 -7995.183} C_VEL
LIN {X 0,Y 462.497,Z 633.601,A -85,B 0,C 180,E1 -7995.76,E2 -7995.76} C_VEL
LIN {X 0,Y 462.046,Z 645.437,A -85,B 0,C 180,E1 -7996.475,E2 -7996.475} C_VEL
LIN {X 0,Y 461.595,Z 657.058,A -85,B 0,C 180,E1 -7997.383,E2 -7997.383} C_VEL
LIN {X 0,Y 461.082,Z 666.946,A -85,B 0,C 180,E1 -7998.348,E2 -7998.348} C_VEL
LIN {X 0,Y 460.624,Z 676.062,A -85,B 0,C 180,E1 -7999.45,E2 -7999.45} C_VEL
LIN {X 0,Y 460.244,Z 684.913,A -85,B 0,C 180,E1 -8000.773,E2 -8000.773} C_VEL
LIN {X 0,Y 459.989,Z 692.002,A -85,B 0,C 180,E1 -8002.096,E2 -8002.096} C_VEL
LIN {X 0,Y 459.786,Z 697.896,A -85,B 0,C 180,E1 -8003.49,E2 -8003.49} C_VEL
LIN {X 0,Y 459.753,Z 702.036,A -85,B 0,C 180,E1 -8004.737,E2 -8004.737} C_VEL
LIN {X 0,Y 459.636,Z 704.353,A -85,B 0,C 180,E1 -8005.615,E2 -8005.615} C_VEL
LIN {X 0,Y 459.676,Z 706.241,A -85,B 0,C 180,E1 -8006.494,E2 -8006.494} C_VEL
LIN {X 0,Y 459.64,Z 707.667,A -85,B 0,C 180,E1 -8007.371,E2 -8007.371} C_VEL
LIN {X 0,Y 459.584,Z 709.285,A -85,B 0,C 180,E1 -8009.124,E2 -8009.124} C_VEL
LIN {X 0,Y 459.611,Z 709.506,A -85,B 0,C 180,E1 -8010,E2 -8010} C_VEL
LIN {X 0,Y 459.629,Z 709.286,A -85,B 0,C 180,E1 -8010.876,E2 -8010.876} C_VEL
LIN {X 0,Y 459.647,Z 707.667,A -85,B 0,C 180,E1 -8012.629,E2 -8012.629} C_VEL
LIN {X 0,Y 459.685,Z 706.242,A -85,B 0,C 180,E1 -8013.506,E2 -8013.506} C_VEL
LIN {X 0,Y 459.698,Z 703.273,A -85,B 0,C 180,E1 -8014.823,E2 -8014.823} C_VEL
LIN {X 0,Y 459.748,Z 699.239,A -85,B 0,C 180,E1 -8016.143,E2 -8016.143} C_VEL
LIN {X 0,Y 459.923,Z 693.012,A -85,B 0,C 180,E1 -8017.684,E2 -8017.684} C_VEL
LIN {X 0,Y 460.239,Z 686.212,A -85,B 0,C 180,E1 -8019.005,E2 -8019.005} C_VEL
LIN {X 0,Y 460.521,Z 679.245,A -85,B 0,C 180,E1 -8020.108,E2 -8020.108} C_VEL
LIN {X 0,Y 460.891,Z 670.817,A -85,B 0,C 180,E1 -8021.211,E2 -8021.211} C_VEL
LIN {X 0,Y 461.405,Z 660.371,A -85,B 0,C 180,E1 -8022.313,E2 -8022.313} C_VEL
LIN {X 0,Y 461.85,Z 650.003,A -85,B 0,C 180,E1 -8023.194,E2 -8023.194} C_VEL
LIN {X 0,Y 462.294,Z 638.542,A -85,B 0,C 180,E1 -8023.966,E2 -8023.966} C_VEL
LIN {X 0,Y 462.751,Z 626.6,A -85,B 0,C 180,E1 -8024.569,E2 -8024.569} C_VEL
LIN {X 0,Y 463.102,Z 613.629,A -85,B 0,C 180,E1 -8025.035,E2 -8025.035} C_VEL
LIN {X 0,Y 463.298,Z 601.19,A -85,B 0,C 180,E1 -8025.31,E2 -8025.31} C_VEL
LIN {X 0,Y 463.846,Z 531.788,A -85,B 0,C 180,E1 -8026.409,E2 -8026.409} C_VEL
LIN {X 0,Y 463.935,Z 511.425,A -85,B 0,C 180,E1 -8026.79,E2 -8026.79} C_VEL
LIN {X 0,Y 461.235,Z 483.686,A -85,B 0,C 180,E1 -8027.46,E2 -8027.46} C_VEL
LIN {X 0,Y 461.878,Z 462.603,A -85,B 0,C 180,E1 -8030.253,E2 -8030.253} C_VEL
LIN {X 0,Y 462.765,Z 440.623,A -85,B 0,C 180,E1 -8033.257,E2 -8033.257} C_VEL
LIN {X 0,Y 463.791,Z 419.633,A -85,B 0,C 180,E1 -8036.218,E2 -8036.218} C_VEL
LIN {X 0,Y 464.389,Z 409.205,A -85,B 0,C 180,E1 -8037.734,E2 -8037.734} C_VEL
LIN {X 0,Y 462.174,Z 397.827,A -85,B 0,C 180,E1 -8039.63,E2 -8039.63} C_VEL
LIN {X 0,Y 460.503,Z 391.222,A -85,B 0,C 180,E1 -8040.859,E2 -8040.859} C_VEL
LIN {X 0,Y 460.501,Z 391.126,A -85,B 0,C 180,E1 -8043.327,E2 -8043.327} C_VEL
LIN {X 0,Y 460.457,Z 391.13,A -85,B 0,C 180,E1 -8046.531,E2 -8046.531} C_VEL
LIN {X 0,Y 460.493,Z 391.127,A -85,B 0,C 180,E1 -8049.867,E2 -8049.867} C_VEL
LIN {X 0,Y 460.46,Z 391.127,A -85,B 0,C 180,E1 -8052.893,E2 -8052.893} C_VEL
LIN {X 0,Y 460.504,Z 391.126,A -85,B 0,C 180,E1 -8055.832,E2 -8055.832} C_VEL
LIN {X 0,Y 460.515,Z 391.119,A -85,B 0,C 180,E1 -8058.987,E2 -8058.987} C_VEL
LIN {X 0,Y 460.488,Z 391.123,A -85,B 0,C 180,E1 -8062.375,E2 -8062.375} C_VEL
LIN {X 0,Y 460.538,Z 391.119,A -85,B 0,C 180,E1 -8065.623,E2 -8065.623} C_VEL
LIN {X 0,Y 460.539,Z 391.117,A -85,B 0,C 180,E1 -8068.745,E2 -8068.745} C_VEL
LIN {X 0,Y 460.553,Z 391.115,A -85,B 0,C 180,E1 -8072.261,E2 -8072.261} C_VEL
LIN {X 0,Y 460.537,Z 391.117,A -85,B 0,C 180,E1 -8074.704,E2 -8074.704} C_VEL
LIN {X 0,Y 460.513,Z 391.125,A -85,B 0,C 180,E1 -8077.571,E2 -8077.571} C_VEL
LIN {X 0,Y 460.571,Z 391.116,A -85,B 0,C 180,E1 -8080.385,E2 -8080.385} C_VEL
LIN {X 0,Y 460.584,Z 391.3,A -85,B 0,C 180,E1 -8082.918,E2 -8082.918} C_VEL
LIN {X 0,Y 460.776,Z 392.21,A -85,B 0,C 180,E1 -8083.058,E2 -8083.058} C_VEL
LIN {X 0,Y 464.733,Z 402.169,A -85,B 0,C 180,E1 -8083.475,E2 -8083.475} C_VEL
LIN {X 0,Y 463.832,Z 475.839,A -85,B 0,C 180,E1 -8084.877,E2 -8084.877} C_VEL
LIN {X 0,Y 463.777,Z 489.625,A -85,B 0,C 180,E1 -8085.324,E2 -8085.324} C_VEL
LIN {X 0,Y 463.606,Z 500.963,A -85,B 0,C 180,E1 -8085.851,E2 -8085.851} C_VEL
LIN {X 0,Y 463.373,Z 511.323,A -85,B 0,C 180,E1 -8086.478,E2 -8086.478} C_VEL
LIN {X 0,Y 463.03,Z 521.887,A -85,B 0,C 180,E1 -8087.286,E2 -8087.286} C_VEL
LIN {X 0,Y 462.599,Z 531.27,A -85,B 0,C 180,E1 -8088.165,E2 -8088.165} C_VEL
LIN {X 0,Y 462.237,Z 540.804,A -85,B 0,C 180,E1 -8089.266,E2 -8089.266} C_VEL
LIN {X 0,Y 461.817,Z 548.59,A -85,B 0,C 180,E1 -8090.363,E2 -8090.363} C_VEL
LIN {X 0,Y 461.54,Z 556.11,A -85,B 0,C 180,E1 -8091.683,E2 -8091.683} C_VEL
LIN {X 0,Y 461.221,Z 562.085,A -85,B 0,C 180,E1 -8092.998,E2 -8092.998} C_VEL
LIN {X 0,Y 460.97,Z 566.771,A -85,B 0,C 180,E1 -8094.313,E2 -8094.313} C_VEL
LIN {X 0,Y 460.667,Z 570.334,A -85,B 0,C 180,E1 -8095.625,E2 -8095.625} C_VEL
LIN {X 0,Y 460.71,Z 572.107,A -85,B 0,C 180,E1 -8096.502,E2 -8096.502} C_VEL
LIN {X 0,Y 460.585,Z 573.455,A -85,B 0,C 180,E1 -8097.376,E2 -8097.376} C_VEL
LIN {X 0,Y 460.528,Z 574.354,A -85,B 0,C 180,E1 -8098.251,E2 -8098.251} C_VEL
LIN {X 0,Y 460.441,Z 574.866,A -85,B 0,C 180,E1 -8099.125,E2 -8099.125} C_VEL
LIN {X 0,Y 460.407,Z 574.974,A -85,B 0,C 180,E1 -8100,E2 -8100} C_VEL
LIN {X 0,Y 460.424,Z 574.628,A -85,B 0,C 180,E1 -8100.875,E2 -8100.875} C_VEL
LIN {X 0,Y 460.347,Z 573.897,A -85,B 0,C 180,E1 -8101.75,E2 -8101.75} C_VEL
LIN {X 0,Y 460.464,Z 572.748,A -85,B 0,C 180,E1 -8102.624,E2 -8102.624} C_VEL
LIN {X 0,Y 460.465,Z 570.23,A -85,B 0,C 180,E1 -8103.938,E2 -8103.938} C_VEL
LIN {X 0,Y 460.575,Z 566.689,A -85,B 0,C 180,E1 -8105.253,E2 -8105.253} C_VEL
LIN {X 0,Y 460.831,Z 562.027,A -85,B 0,C 180,E1 -8106.568,E2 -8106.568} C_VEL
LIN {X 0,Y 461.134,Z 554.967,A -85,B 0,C 180,E1 -8108.104,E2 -8108.104} C_VEL
LIN {X 0,Y 461.416,Z 547.307,A -85,B 0,C 180,E1 -8109.424,E2 -8109.424} C_VEL
LIN {X 0,Y 461.706,Z 539.481,A -85,B 0,C 180,E1 -8110.525,E2 -8110.525} C_VEL
LIN {X 0,Y 462.079,Z 529.915,A -85,B 0,C 180,E1 -8111.626,E2 -8111.626} C_VEL
LIN {X 0,Y 462.468,Z 519.265,A -85,B 0,C 180,E1 -8112.618,E2 -8112.618} C_VEL
LIN {X 0,Y 462.77,Z 507.512,A -85,B 0,C 180,E1 -8113.496,E2 -8113.496} C_VEL
LIN {X 0,Y 463.045,Z 494.736,A -85,B 0,C 180,E1 -8114.223,E2 -8114.223} C_VEL
LIN {X 0,Y 463.301,Z 482.201,A -85,B 0,C 180,E1 -8114.748,E2 -8114.748} C_VEL
LIN {X 0,Y 463.334,Z 469.333,A -85,B 0,C 180,E1 -8115.112,E2 -8115.112} C_VEL
LIN {X 0,Y 464.017,Z 401.831,A -85,B 0,C 180,E1 -8116.298,E2 -8116.298} C_VEL
LIN {X 0,Y 460.772,Z 392.128,A -85,B 0,C 180,E1 -8116.602,E2 -8116.602} C_VEL
LIN {X 0,Y 460.589,Z 391.198,A -85,B 0,C 180,E1 -8116.777,E2 -8116.777} C_VEL
LIN {X 0,Y 460.571,Z 391.114,A -85,B 0,C 180,E1 -8119.616,E2 -8119.616} C_VEL
LIN {X 0,Y 460.514,Z 391.123,A -85,B 0,C 180,E1 -8122.429,E2 -8122.429} C_VEL
LIN {X 0,Y 460.552,Z 391.113,A -85,B 0,C 180,E1 -8125.797,E2 -8125.797} C_VEL
LIN {X 0,Y 460.529,Z 391.113,A -85,B 0,C 180,E1 -8128.235,E2 -8128.235} C_VEL
LIN {X 0,Y 460.523,Z 391.119,A -85,B 0,C 180,E1 -8131.283,E2 -8131.283} C_VEL
LIN {X 0,Y 460.525,Z 391.113,A -85,B 0,C 180,E1 -8134.504,E2 -8134.504} C_VEL
LIN {X 0,Y 460.503,Z 391.116,A -85,B 0,C 180,E1 -8137.623,E2 -8137.623} C_VEL
LIN {X 0,Y 460.538,Z 391.118,A -85,B 0,C 180,E1 -8140.269,E2 -8140.269} C_VEL
LIN {X 0,Y 460.51,Z 391.12,A -85,B 0,C 180,E1 -8143.374,E2 -8143.374} C_VEL
LIN {X 0,Y 460.511,Z 391.125,A -85,B 0,C 180,E1 -8146.626,E2 -8146.626} C_VEL
LIN {X 0,Y 460.536,Z 391.117,A -85,B 0,C 180,E1 -8149.732,E2 -8149.732} C_VEL
LIN {X 0,Y 460.499,Z 391.118,A -85,B 0,C 180,E1 -8152.524,E2 -8152.524} C_VEL
LIN {X 0,Y 460.548,Z 391.113,A -85,B 0,C 180,E1 -8155.624,E2 -8155.624} C_VEL
LIN {X 0,Y 460.54,Z 391.121,A -85,B 0,C 180,E1 -8158.745,E2 -8158.745} C_VEL
LIN {X 0,Y 460.572,Z 391.369,A -85,B 0,C 180,E1 -8159.764,E2 -8159.764} C_VEL
LIN {X 0,Y 464.166,Z 406.354,A -85,B 0,C 180,E1 -8162.006,E2 -8162.006} C_VEL
LIN {X 0,Y 464.887,Z 409.991,A -85,B 0,C 180,E1 -8162.543,E2 -8162.543} C_VEL
LIN {X 0,Y 464.298,Z 429.472,A -85,B 0,C 180,E1 -8165.176,E2 -8165.176} C_VEL
LIN {X 0,Y 464.279,Z 429.737,A -85,B 0,C 180,E1 -8165.211,E2 -8165.211} C_VEL
LIN {X 0,Y 463.393,Z 433.845,A -85,B 0,C 180,E1 -8165.726,E2 -8165.726} C_VEL
LIN {X 0,Y 457.288,Z 447.678,A -85,B 0,C 180,E1 -8167.327,E2 -8167.327} C_VEL
LIN {X 0,Y 456.5,Z 451.799,A -85,B 0,C 180,E1 -8167.851,E2 -8167.851} C_VEL
LIN {X 0,Y 455.658,Z 474.787,A -85,B 0,C 180,E1 -8170.872,E2 -8170.872} C_VEL
LIN {X 0,Y 455.387,Z 488.038,A -85,B 0,C 180,E1 -8172.504,E2 -8172.504} C_VEL
LIN {X 0,Y 457.731,Z 505.51,A -85,B 0,C 180,E1 -8172.887,E2 -8172.887} C_VEL
LIN {X 0,Y 456.885,Z 598.843,A -85,B 0,C 180,E1 -8174.384,E2 -8174.384} C_VEL
LIN {X 0,Y 456.528,Z 612.245,A -85,B 0,C 180,E1 -8174.772,E2 -8174.772} C_VEL
LIN {X 0,Y 456.068,Z 624.786,A -85,B 0,C 180,E1 -8175.327,E2 -8175.327} C_VEL
LIN {X 0,Y 455.568,Z 636.902,A -85,B 0,C 180,E1 -8176.052,E2 -8176.052} C_VEL
LIN {X 0,Y 455.085,Z 648.462,A -85,B 0,C 180,E1 -8176.955,E2 -8176.955} C_VEL
LIN {X 0,Y 454.528,Z 658.645,A -85,B 0,C 180,E1 -8177.952,E2 -8177.952} C_VEL
LIN {X 0,Y 453.927,Z 667.952,A -85,B 0,C 180,E1 -8179.067,E2 -8179.067} C_VEL
LIN {X 0,Y 453.447,Z 676.931,A -85,B 0,C 180,E1 -8180.409,E2 -8180.409} C_VEL
LIN {X 0,Y 453.06,Z 684.14,A -85,B 0,C 180,E1 -8181.75,E2 -8181.75} C_VEL
LIN {X 0,Y 452.866,Z 689.034,A -85,B 0,C 180,E1 -8182.868,E2 -8182.868} C_VEL
LIN {X 0,Y 452.718,Z 693.771,A -85,B 0,C 180,E1 -8184.209,E2 -8184.209} C_VEL
LIN {X 0,Y 452.521,Z 697.399,A -85,B 0,C 180,E1 -8185.546,E2 -8185.546} C_VEL
LIN {X 0,Y 452.504,Z 699.267,A -85,B 0,C 180,E1 -8186.438,E2 -8186.438} C_VEL
LIN {X 0,Y 452.511,Z 700.696,A -85,B 0,C 180,E1 -8187.33,E2 -8187.33} C_VEL
LIN {X 0,Y 452.404,Z 702.316,A -85,B 0,C 180,E1 -8189.11,E2 -8189.11} C_VEL
LIN {X 0,Y 452.407,Z 702.554,A -85,B 0,C 180,E1 -8190,E2 -8190} C_VEL
LIN {X 0,Y 452.404,Z 702.364,A -85,B 0,C 180,E1 -8190.89,E2 -8190.89} C_VEL
LIN {X 0,Y 452.511,Z 700.807,A -85,B 0,C 180,E1 -8192.671,E2 -8192.671} C_VEL
LIN {X 0,Y 452.504,Z 699.44,A -85,B 0,C 180,E1 -8193.562,E2 -8193.562} C_VEL
LIN {X 0,Y 452.578,Z 696.563,A -85,B 0,C 180,E1 -8194.9,E2 -8194.9} C_VEL
LIN {X 0,Y 452.71,Z 691.717,A -85,B 0,C 180,E1 -8196.506,E2 -8196.506} C_VEL
LIN {X 0,Y 452.981,Z 685.619,A -85,B 0,C 180,E1 -8198.027,E2 -8198.027} C_VEL
LIN {X 0,Y 453.325,Z 678.78,A -85,B 0,C 180,E1 -8199.369,E2 -8199.369} C_VEL
LIN {X 0,Y 453.779,Z 670.225,A -85,B 0,C 180,E1 -8200.711,E2 -8200.711} C_VEL
LIN {X 0,Y 454.364,Z 661.467,A -85,B 0,C 180,E1 -8201.827,E2 -8201.827} C_VEL
LIN {X 0,Y 454.911,Z 651.63,A -85,B 0,C 180,E1 -8202.853,E2 -8202.853} C_VEL
LIN {X 0,Y 455.358,Z 641.235,A -85,B 0,C 180,E1 -8203.727,E2 -8203.727} C_VEL
LIN {X 0,Y 455.942,Z 629.473,A -85,B 0,C 180,E1 -8204.506,E2 -8204.506} C_VEL
LIN {X 0,Y 456.363,Z 617.309,A -85,B 0,C 180,E1 -8205.12,E2 -8205.12} C_VEL
LIN {X 0,Y 456.841,Z 604.619,A -85,B 0,C 180,E1 -8205.561,E2 -8205.561} C_VEL
LIN {X 0,Y 457.063,Z 591.793,A -85,B 0,C 180,E1 -8205.839,E2 -8205.839} C_VEL
LIN {X 0,Y 457.672,Z 503.861,A -85,B 0,C 180,E1 -8207.234,E2 -8207.234} C_VEL
LIN {X 0,Y 455.364,Z 487.791,A -85,B 0,C 180,E1 -8207.603,E2 -8207.603} C_VEL
LIN {X 0,Y 455.871,Z 468.485,A -85,B 0,C 180,E1 -8210.038,E2 -8210.038} C_VEL
LIN {X 0,Y 456.876,Z 443.725,A -85,B 0,C 180,E1 -8213.335,E2 -8213.335} C_VEL
LIN {X 0,Y 457.699,Z 424.429,A -85,B 0,C 180,E1 -8215.952,E2 -8215.952} C_VEL
LIN {X 0,Y 458.107,Z 411.939,A -85,B 0,C 180,E1 -8217.651,E2 -8217.651} C_VEL
LIN {X 0,Y 454.53,Z 396.139,A -85,B 0,C 180,E1 -8220.016,E2 -8220.016} C_VEL
LIN {X 0,Y 453.519,Z 392.195,A -85,B 0,C 180,E1 -8220.647,E2 -8220.647} C_VEL
LIN {X 0,Y 453.47,Z 391.996,A -85,B 0,C 180,E1 -8223.914,E2 -8223.914} C_VEL
LIN {X 0,Y 453.439,Z 391.996,A -85,B 0,C 180,E1 -8227.191,E2 -8227.191} C_VEL
LIN {X 0,Y 453.472,Z 391.988,A -85,B 0,C 180,E1 -8230.612,E2 -8230.612} C_VEL
LIN {X 0,Y 453.461,Z 391.985,A -85,B 0,C 180,E1 -8234.222,E2 -8234.222} C_VEL
LIN {X 0,Y 453.44,Z 392.001,A -85,B 0,C 180,E1 -8237.002,E2 -8237.002} C_VEL
LIN {X 0,Y 453.473,Z 391.997,A -85,B 0,C 180,E1 -8239.413,E2 -8239.413} C_VEL
LIN {X 0,Y 453.442,Z 391.994,A -85,B 0,C 180,E1 -8242.809,E2 -8242.809} C_VEL
LIN {X 0,Y 453.469,Z 391.991,A -85,B 0,C 180,E1 -8246.086,E2 -8246.086} C_VEL
LIN {X 0,Y 453.477,Z 391.998,A -85,B 0,C 180,E1 -8249.24,E2 -8249.24} C_VEL
LIN {X 0,Y 453.476,Z 391.995,A -85,B 0,C 180,E1 -8252.293,E2 -8252.293} C_VEL
LIN {X 0,Y 453.49,Z 391.995,A -85,B 0,C 180,E1 -8255.264,E2 -8255.264} C_VEL
LIN {X 0,Y 453.485,Z 391.994,A -85,B 0,C 180,E1 -8258.415,E2 -8258.415} C_VEL
LIN {X 0,Y 453.527,Z 391.986,A -85,B 0,C 180,E1 -8261.009,E2 -8261.009} C_VEL
LIN {X 0,Y 453.524,Z 391.988,A -85,B 0,C 180,E1 -8264.726,E2 -8264.726} C_VEL
LIN {X 0,Y 453.568,Z 391.982,A -85,B 0,C 180,E1 -8267.471,E2 -8267.471} C_VEL
LIN {X 0,Y 453.563,Z 391.983,A -85,B 0,C 180,E1 -8271.086,E2 -8271.086} C_VEL
LIN {X 0,Y 453.64,Z 391.973,A -85,B 0,C 180,E1 -8273.774,E2 -8273.774} C_VEL
LIN {X 0,Y 453.705,Z 391.963,A -85,B 0,C 180,E1 -8277.336,E2 -8277.336} C_VEL
LIN {X 0,Y 453.771,Z 391.958,A -85,B 0,C 180,E1 -8280,E2 -8280} C_VEL
LIN {X 0,Y 453.706,Z 391.953,A -85,B 0,C 180,E1 -8282.663,E2 -8282.663} C_VEL
LIN {X 0,Y 453.639,Z 391.976,A -85,B 0,C 180,E1 -8286.226,E2 -8286.226} C_VEL
LIN {X 0,Y 453.561,Z 391.975,A -85,B 0,C 180,E1 -8288.914,E2 -8288.914} C_VEL
LIN {X 0,Y 453.568,Z 391.983,A -85,B 0,C 180,E1 -8292.529,E2 -8292.529} C_VEL
LIN {X 0,Y 453.488,Z 391.983,A -85,B 0,C 180,E1 -8296.198,E2 -8296.198} C_VEL
LIN {X 0,Y 453.489,Z 391.992,A -85,B 0,C 180,E1 -8299.027,E2 -8299.027} C_VEL
LIN {X 0,Y 453.474,Z 391.992,A -85,B 0,C 180,E1 -8301.836,E2 -8301.836} C_VEL
LIN {X 0,Y 453.465,Z 391.994,A -85,B 0,C 180,E1 -8304.737,E2 -8304.737} C_VEL
LIN {X 0,Y 453.463,Z 391.994,A -85,B 0,C 180,E1 -8307.942,E2 -8307.942} C_VEL
LIN {X 0,Y 453.459,Z 391.995,A -85,B 0,C 180,E1 -8310.761,E2 -8310.761} C_VEL
LIN {X 0,Y 453.467,Z 391.993,A -85,B 0,C 180,E1 -8313.914,E2 -8313.914} C_VEL
LIN {X 0,Y 453.436,Z 392.001,A -85,B 0,C 180,E1 -8317.191,E2 -8317.191} C_VEL
LIN {X 0,Y 453.466,Z 391.973,A -85,B 0,C 180,E1 -8320.612,E2 -8320.612} C_VEL
LIN {X 0,Y 453.478,Z 391.995,A -85,B 0,C 180,E1 -8324.527,E2 -8324.527} C_VEL
LIN {X 0,Y 453.432,Z 391.983,A -85,B 0,C 180,E1 -8328.072,E2 -8328.072} C_VEL
LIN {X 0,Y 453.425,Z 391.999,A -85,B 0,C 180,E1 -8330.804,E2 -8330.804} C_VEL
LIN {X 0,Y 453.44,Z 392.006,A -85,B 0,C 180,E1 -8333.915,E2 -8333.915} C_VEL
LIN {X 0,Y 453.466,Z 392,A -85,B 0,C 180,E1 -8336.816,E2 -8336.816} C_VEL
LIN {X 0,Y 453.48,Z 392.195,A -85,B 0,C 180,E1 -8338.877,E2 -8338.877} C_VEL
LIN {X 0,Y 457.8,Z 410.882,A -85,B 0,C 180,E1 -8341.831,E2 -8341.831} C_VEL
LIN {X 0,Y 457.794,Z 416.097,A -85,B 0,C 180,E1 -8342.577,E2 -8342.577} C_VEL
LIN {X 0,Y 456.664,Z 436.696,A -85,B 0,C 180,E1 -8345.447,E2 -8345.447} C_VEL
LIN {X 0,Y 455.571,Z 458.923,A -85,B 0,C 180,E1 -8348.507,E2 -8348.507} C_VEL
LIN {X 0,Y 454.637,Z 482.783,A -85,B 0,C 180,E1 -8351.758,E2 -8351.758} C_VEL
LIN {X 0,Y 454.461,Z 488.364,A -85,B 0,C 180,E1 -8352.479,E2 -8352.479} C_VEL
LIN {X 0,Y 457.203,Z 514.855,A -85,B 0,C 180,E1 -8353.072,E2 -8353.072} C_VEL
LIN {X 0,Y 456.401,Z 607.234,A -85,B 0,C 180,E1 -8354.567,E2 -8354.567} C_VEL
LIN {X 0,Y 456.061,Z 619.658,A -85,B 0,C 180,E1 -8354.927,E2 -8354.927} C_VEL
LIN {X 0,Y 455.642,Z 632.473,A -85,B 0,C 180,E1 -8355.484,E2 -8355.484} C_VEL
LIN {X 0,Y 455.219,Z 643.823,A -85,B 0,C 180,E1 -8356.155,E2 -8356.155} C_VEL
LIN {X 0,Y 454.734,Z 654.895,A -85,B 0,C 180,E1 -8357.001,E2 -8357.001} C_VEL
LIN {X 0,Y 454.127,Z 665.859,A -85,B 0,C 180,E1 -8358.054,E2 -8358.054} C_VEL
LIN {X 0,Y 453.758,Z 674.355,A -85,B 0,C 180,E1 -8359.063,E2 -8359.063} C_VEL
LIN {X 0,Y 453.34,Z 682.156,A -85,B 0,C 180,E1 -8360.181,E2 -8360.181} C_VEL
LIN {X 0,Y 453.018,Z 689.745,A -85,B 0,C 180,E1 -8361.525,E2 -8361.525} C_VEL
LIN {X 0,Y 452.761,Z 695.832,A -85,B 0,C 180,E1 -8362.866,E2 -8362.866} C_VEL
LIN {X 0,Y 452.672,Z 700.636,A -85,B 0,C 180,E1 -8364.208,E2 -8364.208} C_VEL
LIN {X 0,Y 452.554,Z 704.3,A -85,B 0,C 180,E1 -8365.546,E2 -8365.546} C_VEL
LIN {X 0,Y 452.571,Z 706.188,A -85,B 0,C 180,E1 -8366.439,E2 -8366.439} C_VEL
LIN {X 0,Y 452.563,Z 707.613,A -85,B 0,C 180,E1 -8367.33,E2 -8367.33} C_VEL
LIN {X 0,Y 452.487,Z 709.231,A -85,B 0,C 180,E1 -8369.11,E2 -8369.11} C_VEL
LIN {X 0,Y 452.511,Z 709.452,A -85,B 0,C 180,E1 -8370,E2 -8370} C_VEL
LIN {X 0,Y 452.53,Z 709.231,A -85,B 0,C 180,E1 -8370.89,E2 -8370.89} C_VEL
LIN {X 0,Y 452.57,Z 707.614,A -85,B 0,C 180,E1 -8372.67,E2 -8372.67} C_VEL
LIN {X 0,Y 452.581,Z 706.188,A -85,B 0,C 180,E1 -8373.561,E2 -8373.561} C_VEL
LIN {X 0,Y 452.628,Z 703.22,A -85,B 0,C 180,E1 -8374.899,E2 -8374.899} C_VEL
LIN {X 0,Y 452.709,Z 698.225,A -85,B 0,C 180,E1 -8376.506,E2 -8376.506} C_VEL
LIN {X 0,Y 452.94,Z 691.953,A -85,B 0,C 180,E1 -8378.027,E2 -8378.027} C_VEL
LIN {X 0,Y 453.22,Z 684.866,A -85,B 0,C 180,E1 -8379.371,E2 -8379.371} C_VEL
LIN {X 0,Y 453.625,Z 676.004,A -85,B 0,C 180,E1 -8380.714,E2 -8380.714} C_VEL
LIN {X 0,Y 454.137,Z 666.883,A -85,B 0,C 180,E1 -8381.832,E2 -8381.832} C_VEL
LIN {X 0,Y 454.696,Z 656.24,A -85,B 0,C 180,E1 -8382.879,E2 -8382.879} C_VEL
LIN {X 0,Y 455.15,Z 645.386,A -85,B 0,C 180,E1 -8383.733,E2 -8383.733} C_VEL
LIN {X 0,Y 455.622,Z 633.549,A -85,B 0,C 180,E1 -8384.459,E2 -8384.459} C_VEL
LIN {X 0,Y 456.053,Z 620.363,A -85,B 0,C 180,E1 -8385.045,E2 -8385.045} C_VEL
LIN {X 0,Y 456.415,Z 607.161,A -85,B 0,C 180,E1 -8385.432,E2 -8385.432} C_VEL
LIN {X 0,Y 457.043,Z 532.544,A -85,B 0,C 180,E1 -8386.651,E2 -8386.651} C_VEL
LIN {X 0,Y 457.181,Z 512.144,A -85,B 0,C 180,E1 -8387.046,E2 -8387.046} C_VEL
LIN {X 0,Y 454.313,Z 482.963,A -85,B 0,C 180,E1 -8387.766,E2 -8387.766} C_VEL
LIN {X 0,Y 454.296,Z 481.674,A -85,B 0,C 180,E1 -8387.863,E2 -8387.863} C_VEL
LIN {X 0,Y 455.124,Z 456.71,A -85,B 0,C 180,E1 -8391.278,E2 -8391.278} C_VEL
LIN {X 0,Y 456.141,Z 434.972,A -85,B 0,C 180,E1 -8394.34,E2 -8394.34} C_VEL
LIN {X 0,Y 457.399,Z 414.85,A -85,B 0,C 180,E1 -8397.277,E2 -8397.277} C_VEL
LIN {X 0,Y 457.55,Z 410.498,A -85,B 0,C 180,E1 -8397.936,E2 -8397.936} C_VEL
LIN {X 0,Y 455.267,Z 399.186,A -85,B 0,C 180,E1 -8399.884,E2 -8399.884} C_VEL
LIN {X 0,Y 453.469,Z 392.109,A -85,B 0,C 180,E1 -8401.246,E2 -8401.246} C_VEL
LIN {X 0,Y 453.453,Z 392.005,A -85,B 0,C 180,E1 -8403.915,E2 -8403.915} C_VEL
LIN {X 0,Y 453.434,Z 392.004,A -85,B 0,C 180,E1 -8407.192,E2 -8407.192} C_VEL
LIN {X 0,Y 453.465,Z 391.998,A -85,B 0,C 180,E1 -8410.612,E2 -8410.612} C_VEL
LIN {X 0,Y 453.482,Z 391.996,A -85,B 0,C 180,E1 -8414.528,E2 -8414.528} C_VEL
LIN {X 0,Y 453.437,Z 392.002,A -85,B 0,C 180,E1 -8418.071,E2 -8418.071} C_VEL
LIN {X 0,Y 453.444,Z 392,A -85,B 0,C 180,E1 -8420.801,E2 -8420.801} C_VEL
LIN {X 0,Y 453.449,Z 392.002,A -85,B 0,C 180,E1 -8423.917,E2 -8423.917} C_VEL
LIN {X 0,Y 453.481,Z 391.999,A -85,B 0,C 180,E1 -8427.151,E2 -8427.151} C_VEL
LIN {X 0,Y 453.469,Z 391.998,A -85,B 0,C 180,E1 -8430.268,E2 -8430.268} C_VEL
LIN {X 0,Y 453.473,Z 392,A -85,B 0,C 180,E1 -8433.292,E2 -8433.292} C_VEL
LIN {X 0,Y 453.496,Z 391.996,A -85,B 0,C 180,E1 -8436.238,E2 -8436.238} C_VEL
LIN {X 0,Y 453.485,Z 392,A -85,B 0,C 180,E1 -8439.118,E2 -8439.118} C_VEL
LIN {X 0,Y 453.539,Z 392.026,A -85,B 0,C 180,E1 -8442.459,E2 -8442.459} C_VEL
LIN {X 0,Y 453.622,Z 392.618,A -85,B 0,C 180,E1 -8442.671,E2 -8442.671} C_VEL
LIN {X 0,Y 454.827,Z 395.766,A -85,B 0,C 180,E1 -8442.852,E2 -8442.852} C_VEL
LIN {X 0,Y 458.092,Z 403.829,A -85,B 0,C 180,E1 -8443.186,E2 -8443.186} C_VEL
LIN {X 0,Y 457.114,Z 477.756,A -85,B 0,C 180,E1 -8444.649,E2 -8444.649} C_VEL
LIN {X 0,Y 457.032,Z 491.284,A -85,B 0,C 180,E1 -8445.102,E2 -8445.102} C_VEL
LIN {X 0,Y 456.833,Z 502.501,A -85,B 0,C 180,E1 -8445.637,E2 -8445.637} C_VEL
LIN {X 0,Y 456.526,Z 514.341,A -85,B 0,C 180,E1 -8446.386,E2 -8446.386} C_VEL
LIN {X 0,Y 456.076,Z 525.814,A -85,B 0,C 180,E1 -8447.315,E2 -8447.315} C_VEL
LIN {X 0,Y 455.7,Z 534.686,A -85,B 0,C 180,E1 -8448.209,E2 -8448.209} C_VEL
LIN {X 0,Y 455.334,Z 543.736,A -85,B 0,C 180,E1 -8449.326,E2 -8449.326} C_VEL
LIN {X 0,Y 454.881,Z 551.159,A -85,B 0,C 180,E1 -8450.439,E2 -8450.439} C_VEL
LIN {X 0,Y 454.543,Z 558.054,A -85,B 0,C 180,E1 -8451.71,E2 -8451.71} C_VEL
LIN {X 0,Y 454.27,Z 563.256,A -85,B 0,C 180,E1 -8452.89,E2 -8452.89} C_VEL
LIN {X 0,Y 454.023,Z 567.923,A -85,B 0,C 180,E1 -8454.225,E2 -8454.225} C_VEL
LIN {X 0,Y 453.68,Z 571.471,A -85,B 0,C 180,E1 -8455.558,E2 -8455.558} C_VEL
LIN {X 0,Y 453.728,Z 573.229,A -85,B 0,C 180,E1 -8456.448,E2 -8456.448} C_VEL
LIN {X 0,Y 453.591,Z 574.553,A -85,B 0,C 180,E1 -8457.336,E2 -8457.336} C_VEL
LIN {X 0,Y 453.515,Z 575.44,A -85,B 0,C 180,E1 -8458.224,E2 -8458.224} C_VEL
LIN {X 0,Y 453.423,Z 575.932,A -85,B 0,C 180,E1 -8459.112,E2 -8459.112} C_VEL
LIN {X 0,Y 453.385,Z 576.011,A -85,B 0,C 180,E1 -8460,E2 -8460} C_VEL
LIN {X 0,Y 453.402,Z 575.637,A -85,B 0,C 180,E1 -8460.888,E2 -8460.888} C_VEL
LIN {X 0,Y 453.324,Z 574.883,A -85,B 0,C 180,E1 -8461.777,E2 -8461.777} C_VEL
LIN {X 0,Y 453.445,Z 573.703,A -85,B 0,C 180,E1 -8462.665,E2 -8462.665} C_VEL
LIN {X 0,Y 453.437,Z 571.137,A -85,B 0,C 180,E1 -8464,E2 -8464} C_VEL
LIN {X 0,Y 453.571,Z 567.54,A -85,B 0,C 180,E1 -8465.334,E2 -8465.334} C_VEL
LIN {X 0,Y 453.905,Z 561.92,A -85,B 0,C 180,E1 -8466.882,E2 -8466.882} C_VEL
LIN {X 0,Y 454.143,Z 555.666,A -85,B 0,C 180,E1 -8468.23,E2 -8468.23} C_VEL
LIN {X 0,Y 454.43,Z 547.925,A -85,B 0,C 180,E1 -8469.57,E2 -8469.57} C_VEL
LIN {X 0,Y 454.751,Z 540,A -85,B 0,C 180,E1 -8470.688,E2 -8470.688} C_VEL
LIN {X 0,Y 455.145,Z 529.204,A -85,B 0,C 180,E1 -8471.919,E2 -8471.919} C_VEL
LIN {X 0,Y 455.584,Z 518.182,A -85,B 0,C 180,E1 -8472.925,E2 -8472.925} C_VEL
LIN {X 0,Y 455.845,Z 506.675,A -85,B 0,C 180,E1 -8473.758,E2 -8473.758} C_VEL
LIN {X 0,Y 456.156,Z 494.468,A -85,B 0,C 180,E1 -8474.442,E2 -8474.442} C_VEL
LIN {X 0,Y 456.403,Z 481.43,A -85,B 0,C 180,E1 -8474.976,E2 -8474.976} C_VEL
LIN {X 0,Y 456.434,Z 467.45,A -85,B 0,C 180,E1 -8475.346,E2 -8475.346} C_VEL
LIN {X 0,Y 456.999,Z 402.689,A -85,B 0,C 180,E1 -8476.512,E2 -8476.512} C_VEL
LIN {X 0,Y 453.71,Z 392.901,A -85,B 0,C 180,E1 -8476.824,E2 -8476.824} C_VEL
LIN {X 0,Y 453.551,Z 392.052,A -85,B 0,C 180,E1 -8477.008,E2 -8477.008} C_VEL
LIN {X 0,Y 453.507,Z 391.994,A -85,B 0,C 180,E1 -8479.934,E2 -8479.934} C_VEL
LIN {X 0,Y 453.482,Z 392,A -85,B 0,C 180,E1 -8482.796,E2 -8482.796} C_VEL
LIN {X 0,Y 453.5,Z 391.992,A -85,B 0,C 180,E1 -8485.993,E2 -8485.993} C_VEL
LIN {X 0,Y 453.495,Z 391.988,A -85,B 0,C 180,E1 -8488.713,E2 -8488.713} C_VEL
LIN {X 0,Y 453.466,Z 391.996,A -85,B 0,C 180,E1 -8491.8,E2 -8491.8} C_VEL
LIN {X 0,Y 453.478,Z 391.998,A -85,B 0,C 180,E1 -8494.99,E2 -8494.99} C_VEL
LIN {X 0,Y 453.465,Z 391.994,A -85,B 0,C 180,E1 -8498.312,E2 -8498.312} C_VEL
LIN {X 0,Y 453.495,Z 391.999,A -85,B 0,C 180,E1 -8500.609,E2 -8500.609} C_VEL
LIN {X 0,Y 453.462,Z 392.001,A -85,B 0,C 180,E1 -8504.222,E2 -8504.222} C_VEL
LIN {X 0,Y 453.45,Z 392,A -85,B 0,C 180,E1 -8507.003,E2 -8507.003} C_VEL
LIN {X 0,Y 453.496,Z 391.994,A -85,B 0,C 180,E1 -8509.409,E2 -8509.409} C_VEL
LIN {X 0,Y 453.451,Z 392.001,A -85,B 0,C 180,E1 -8512.81,E2 -8512.81} C_VEL
LIN {X 0,Y 453.479,Z 391.997,A -85,B 0,C 180,E1 -8516.087,E2 -8516.087} C_VEL
LIN {X 0,Y 453.531,Z 392.155,A -85,B 0,C 180,E1 -8519.443,E2 -8519.443} C_VEL
LIN {X 0,Y 457.226,Z 407.551,A -85,B 0,C 180,E1 -8521.793,E2 -8521.793} C_VEL
LIN {X 0,Y 458.11,Z 412.992,A -85,B 0,C 180,E1 -8522.597,E2 -8522.597} C_VEL
LIN {X 0,Y 457.167,Z 435.995,A -85,B 0,C 180,E1 -8525.718,E2 -8525.718} C_VEL
LIN {X 0,Y 456.5,Z 451.799,A -85,B 0,C 180,E1 -8527.851,E2 -8527.851} C_VEL
LIN {X 0,Y 455.705,Z 455.932,A -85,B 0,C 180,E1 -8528.372,E2 -8528.372} C_VEL
LIN {X 0,Y 449.602,Z 469.962,A -85,B 0,C 180,E1 -8529.978,E2 -8529.978} C_VEL
LIN {X 0,Y 448.796,Z 474.172,A -85,B 0,C 180,E1 -8530.501,E2 -8530.501} C_VEL
LIN {X 0,Y 448.509,Z 488.083,A -85,B 0,C 180,E1 -8532.23,E2 -8532.23} C_VEL
LIN {X 0,Y 450.933,Z 505.319,A -85,B 0,C 180,E1 -8532.619,E2 -8532.619} C_VEL
LIN {X 0,Y 450.059,Z 598.825,A -85,B 0,C 180,E1 -8534.141,E2 -8534.141} C_VEL
LIN {X 0,Y 449.699,Z 612.262,A -85,B 0,C 180,E1 -8534.535,E2 -8534.535} C_VEL
LIN {X 0,Y 449.208,Z 624.818,A -85,B 0,C 180,E1 -8535.098,E2 -8535.098} C_VEL
LIN {X 0,Y 448.671,Z 636.937,A -85,B 0,C 180,E1 -8535.833,E2 -8535.833} C_VEL
LIN {X 0,Y 448.193,Z 647.379,A -85,B 0,C 180,E1 -8536.647,E2 -8536.647} C_VEL
LIN {X 0,Y 447.629,Z 657.658,A -85,B 0,C 180,E1 -8537.648,E2 -8537.648} C_VEL
LIN {X 0,Y 447.052,Z 666.269,A -85,B 0,C 180,E1 -8538.667,E2 -8538.667} C_VEL
LIN {X 0,Y 446.494,Z 675.647,A -85,B 0,C 180,E1 -8540.029,E2 -8540.029} C_VEL
LIN {X 0,Y 446.077,Z 683.103,A -85,B 0,C 180,E1 -8541.392,E2 -8541.392} C_VEL
LIN {X 0,Y 445.786,Z 689.088,A -85,B 0,C 180,E1 -8542.754,E2 -8542.754} C_VEL
LIN {X 0,Y 445.646,Z 693.825,A -85,B 0,C 180,E1 -8544.117,E2 -8544.117} C_VEL
LIN {X 0,Y 445.446,Z 697.454,A -85,B 0,C 180,E1 -8545.475,E2 -8545.475} C_VEL
LIN {X 0,Y 445.405,Z 699.321,A -85,B 0,C 180,E1 -8546.381,E2 -8546.381} C_VEL
LIN {X 0,Y 445.437,Z 700.75,A -85,B 0,C 180,E1 -8547.287,E2 -8547.287} C_VEL
LIN {X 0,Y 445.316,Z 702.37,A -85,B 0,C 180,E1 -8549.096,E2 -8549.096} C_VEL
LIN {X 0,Y 445.316,Z 702.608,A -85,B 0,C 180,E1 -8550,E2 -8550} C_VEL
LIN {X 0,Y 445.316,Z 702.418,A -85,B 0,C 180,E1 -8550.904,E2 -8550.904} C_VEL
LIN {X 0,Y 445.437,Z 700.861,A -85,B 0,C 180,E1 -8552.713,E2 -8552.713} C_VEL
LIN {X 0,Y 445.405,Z 699.493,A -85,B 0,C 180,E1 -8553.619,E2 -8553.619} C_VEL
LIN {X 0,Y 445.513,Z 696.615,A -85,B 0,C 180,E1 -8554.978,E2 -8554.978} C_VEL
LIN {X 0,Y 445.619,Z 692.196,A -85,B 0,C 180,E1 -8556.487,E2 -8556.487} C_VEL
LIN {X 0,Y 445.93,Z 685.668,A -85,B 0,C 180,E1 -8558.155,E2 -8558.155} C_VEL
LIN {X 0,Y 446.296,Z 678.827,A -85,B 0,C 180,E1 -8559.518,E2 -8559.518} C_VEL
LIN {X 0,Y 446.78,Z 670.269,A -85,B 0,C 180,E1 -8560.881,E2 -8560.881} C_VEL
LIN {X 0,Y 447.409,Z 661.508,A -85,B 0,C 180,E1 -8562.013,E2 -8562.013} C_VEL
LIN {X 0,Y 447.963,Z 652.057,A -85,B 0,C 180,E1 -8563.017,E2 -8563.017} C_VEL
LIN {X 0,Y 448.439,Z 641.264,A -85,B 0,C 180,E1 -8563.943,E2 -8563.943} C_VEL
LIN {X 0,Y 449.085,Z 629.493,A -85,B 0,C 180,E1 -8564.733,E2 -8564.733} C_VEL
LIN {X 0,Y 449.528,Z 617.312,A -85,B 0,C 180,E1 -8565.356,E2 -8565.356} C_VEL
LIN {X 0,Y 450.008,Z 604.588,A -85,B 0,C 180,E1 -8565.803,E2 -8565.803} C_VEL
LIN {X 0,Y 450.242,Z 591.686,A -85,B 0,C 180,E1 -8566.085,E2 -8566.085} C_VEL
LIN {X 0,Y 450.831,Z 504.156,A -85,B 0,C 180,E1 -8567.497,E2 -8567.497} C_VEL
LIN {X 0,Y 448.473,Z 487.769,A -85,B 0,C 180,E1 -8567.882,E2 -8567.882} C_VEL
LIN {X 0,Y 449.137,Z 466.394,A -85,B 0,C 180,E1 -8570.615,E2 -8570.615} C_VEL
LIN {X 0,Y 450.132,Z 441.637,A -85,B 0,C 180,E1 -8573.951,E2 -8573.951} C_VEL
LIN {X 0,Y 451.1,Z 420.396,A -85,B 0,C 180,E1 -8576.86,E2 -8576.86} C_VEL
LIN {X 0,Y 451.206,Z 413.17,A -85,B 0,C 180,E1 -8577.858,E2 -8577.858} C_VEL
LIN {X 0,Y 447.555,Z 397.332,A -85,B 0,C 180,E1 -8580.268,E2 -8580.268} C_VEL
LIN {X 0,Y 446.473,Z 393.027,A -85,B 0,C 180,E1 -8580.967,E2 -8580.967} C_VEL
LIN {X 0,Y 446.449,Z 392.871,A -85,B 0,C 180,E1 -8583.454,E2 -8583.454} C_VEL
LIN {X 0,Y 446.395,Z 392.872,A -85,B 0,C 180,E1 -8586.746,E2 -8586.746} C_VEL
LIN {X 0,Y 446.4,Z 392.869,A -85,B 0,C 180,E1 -8590.203,E2 -8590.203} C_VEL
LIN {X 0,Y 446.388,Z 392.874,A -85,B 0,C 180,E1 -8593.595,E2 -8593.595} C_VEL
LIN {X 0,Y 446.396,Z 392.878,A -85,B 0,C 180,E1 -8596.404,E2 -8596.404} C_VEL
LIN {X 0,Y 446.401,Z 392.88,A -85,B 0,C 180,E1 -8599.797,E2 -8599.797} C_VEL
LIN {X 0,Y 446.398,Z 392.874,A -85,B 0,C 180,E1 -8603.254,E2 -8603.254} C_VEL
LIN {X 0,Y 446.452,Z 392.862,A -85,B 0,C 180,E1 -8606.566,E2 -8606.566} C_VEL
LIN {X 0,Y 446.432,Z 392.872,A -85,B 0,C 180,E1 -8609.98,E2 -8609.98} C_VEL
LIN {X 0,Y 446.396,Z 392.876,A -85,B 0,C 180,E1 -8612.834,E2 -8612.834} C_VEL
LIN {X 0,Y 446.428,Z 392.868,A -85,B 0,C 180,E1 -8615.935,E2 -8615.935} C_VEL
LIN {X 0,Y 446.457,Z 392.869,A -85,B 0,C 180,E1 -8618.773,E2 -8618.773} C_VEL
LIN {X 0,Y 446.444,Z 392.866,A -85,B 0,C 180,E1 -8621.649,E2 -8621.649} C_VEL
LIN {X 0,Y 446.464,Z 392.868,A -85,B 0,C 180,E1 -8624.478,E2 -8624.478} C_VEL
LIN {X 0,Y 446.52,Z 392.861,A -85,B 0,C 180,E1 -8627.384,E2 -8627.384} C_VEL
LIN {X 0,Y 446.513,Z 392.86,A -85,B 0,C 180,E1 -8630.944,E2 -8630.944} C_VEL
LIN {X 0,Y 446.61,Z 392.85,A -85,B 0,C 180,E1 -8633.676,E2 -8633.676} C_VEL
LIN {X 0,Y 446.655,Z 392.84,A -85,B 0,C 180,E1 -8637.294,E2 -8637.294} C_VEL
LIN {X 0,Y 446.721,Z 392.837,A -85,B 0,C 180,E1 -8640,E2 -8640} C_VEL
LIN {X 0,Y 446.655,Z 392.83,A -85,B 0,C 180,E1 -8642.706,E2 -8642.706} C_VEL
LIN {X 0,Y 446.609,Z 392.851,A -85,B 0,C 180,E1 -8646.324,E2 -8646.324} C_VEL
LIN {X 0,Y 446.512,Z 392.854,A -85,B 0,C 180,E1 -8649.056,E2 -8649.056} C_VEL
LIN {X 0,Y 446.525,Z 392.86,A -85,B 0,C 180,E1 -8652.73,E2 -8652.73} C_VEL
LIN {X 0,Y 446.432,Z 392.86,A -85,B 0,C 180,E1 -8656.461,E2 -8656.461} C_VEL
LIN {X 0,Y 446.43,Z 392.873,A -85,B 0,C 180,E1 -8659.305,E2 -8659.305} C_VEL
LIN {X 0,Y 446.415,Z 392.866,A -85,B 0,C 180,E1 -8662.2,E2 -8662.2} C_VEL
LIN {X 0,Y 446.416,Z 392.873,A -85,B 0,C 180,E1 -8665.155,E2 -8665.155} C_VEL
LIN {X 0,Y 446.419,Z 392.867,A -85,B 0,C 180,E1 -8668.183,E2 -8668.183} C_VEL
LIN {X 0,Y 446.411,Z 392.875,A -85,B 0,C 180,E1 -8671.301,E2 -8671.301} C_VEL
LIN {X 0,Y 446.422,Z 392.868,A -85,B 0,C 180,E1 -8674.524,E2 -8674.524} C_VEL
LIN {X 0,Y 446.396,Z 392.876,A -85,B 0,C 180,E1 -8678.075,E2 -8678.075} C_VEL
LIN {X 0,Y 446.396,Z 392.85,A -85,B 0,C 180,E1 -8681.395,E2 -8681.395} C_VEL
LIN {X 0,Y 446.419,Z 392.874,A -85,B 0,C 180,E1 -8685.108,E2 -8685.108} C_VEL
LIN {X 0,Y 446.396,Z 392.854,A -85,B 0,C 180,E1 -8688.605,E2 -8688.605} C_VEL
LIN {X 0,Y 446.389,Z 392.884,A -85,B 0,C 180,E1 -8692.119,E2 -8692.119} C_VEL
LIN {X 0,Y 446.413,Z 392.88,A -85,B 0,C 180,E1 -8695.475,E2 -8695.475} C_VEL
LIN {X 0,Y 446.43,Z 393.059,A -85,B 0,C 180,E1 -8698.614,E2 -8698.614} C_VEL
LIN {X 0,Y 450.73,Z 411.59,A -85,B 0,C 180,E1 -8701.603,E2 -8701.603} C_VEL
LIN {X 0,Y 450.998,Z 415.104,A -85,B 0,C 180,E1 -8702.128,E2 -8702.128} C_VEL
LIN {X 0,Y 449.8,Z 435.734,A -85,B 0,C 180,E1 -8705.047,E2 -8705.047} C_VEL
LIN {X 0,Y 448.71,Z 457.952,A -85,B 0,C 180,E1 -8708.161,E2 -8708.161} C_VEL
LIN {X 0,Y 447.583,Z 483.502,A -85,B 0,C 180,E1 -8711.697,E2 -8711.697} C_VEL
LIN {X 0,Y 447.46,Z 487.691,A -85,B 0,C 180,E1 -8712.224,E2 -8712.224} C_VEL
LIN {X 0,Y 450.362,Z 514.899,A -85,B 0,C 180,E1 -8712.835,E2 -8712.835} C_VEL
LIN {X 0,Y 449.577,Z 607.276,A -85,B 0,C 180,E1 -8714.327,E2 -8714.327} C_VEL
LIN {X 0,Y 449.193,Z 620.412,A -85,B 0,C 180,E1 -8714.72,E2 -8714.72} C_VEL
LIN {X 0,Y 448.73,Z 633.564,A -85,B 0,C 180,E1 -8715.313,E2 -8715.313} C_VEL
LIN {X 0,Y 448.225,Z 645.377,A -85,B 0,C 180,E1 -8716.05,E2 -8716.05} C_VEL
LIN {X 0,Y 447.744,Z 655.792,A -85,B 0,C 180,E1 -8716.879,E2 -8716.879} C_VEL
LIN {X 0,Y 447.12,Z 666.862,A -85,B 0,C 180,E1 -8717.979,E2 -8717.979} C_VEL
LIN {X 0,Y 446.623,Z 675.972,A -85,B 0,C 180,E1 -8719.115,E2 -8719.115} C_VEL
LIN {X 0,Y 446.19,Z 684.818,A -85,B 0,C 180,E1 -8720.48,E2 -8720.48} C_VEL
